99: (* normal operation *)
	(* only if input changes for an equivalent of min_ontime then change the output *)
	(* if there is a directional change then wait until last step is finished *)
	IF in < TIME_TO_REAL(min_ontime)/TIME_TO_REAL(max_runtime)/2 THEN val := 0;
	ELSIF in > 1 - TIME_TO_REAL(min_ontime)/TIME_TO_REAL(max_runtime)/2 THEN val := 1;
	ELSIF differ(LIMIT(0,in,1), val, TIME_TO_REAL(min_ontime) / TIME_TO_REAL(max_runtime)) OR in = 0 OR in = 1 THEN
		IF in < val AND NOT out1 THEN val := in;
		ELSIF in > val AND NOT out2 THEN val := in;
		END_IF;
	END_IF;

END_CASE;

(* output ramp generator *)
rout(in := val);
out1 := rout.busy AND rout.UD;
out2 := rout.busy AND NOT rout.UD;
pos := rout.out;

(* set the busy output and if busy goes low, then set the last time in order to check for min_offtime *)
IF NOT busy AND rout.busy THEN
	last := tn;
ELSIF busy AND NOT rout.busy THEN
	cal_timer := cal_timer + tx;
	last := tn;
END_IF;
busy := rout.busy;



(* revision history

19.10.2006	rev 1.1
	added security checks for end_switch to avoid overrun of the end_switch, hans

23.1.2007		rev 1.2
	deleted unused variables force_on and force_off

15.9.2007	hm	rev 1.3
	replaced Time() with T_PLC_MS for compatibility and performance reasons

*)

END_FUNCTION_BLOCK

// POUs/Mathematical/DIFFER
FUNCTION DIFFER : BOOL
VAR_INPUT
	in1 : REAL;
	in2 : REAL;
	X : REAL;
END_VAR


(*
version 1.1	16 mar 2008
programmer 	hugo
tested by		tobias

this function checks if in1 differs more then x from in2
the output is true if abs(in1-in2) > X

*)

DIFFER := ABS(in1 - in2) > X;

(* revision history
hm		8. oct 2006		rev 1.0
	original version

hm		16. mar 2008	rev 1.1
	improverd code for performance

*)

END_FUNCTION

// POUs/Time&Date/MULTIME
FUNCTION MULTIME : TIME
VAR_INPUT
	t : TIME;
	M : REAL;
END_VAR


(*
version 1.1	14 mar 2008
programmer 	hugo
tested by		tobias

multiplies a time by a real number and returns a time
*)

MULTIME := DWORD_TO_TIME(REAL_TO_DWORD(DWORD_TO_REAL(TIME_TO_DWORD(t))*M));

(* revision history
hm		2. oct 2006	rev 1.0
	original version

hm		14. mar 2008	rev 1.1
	rounded the result after the last digit

*)

END_FUNCTION

// POUs/Engineering/measurements/CALIBRATE
FUNCTION_BLOCK CALIBRATE
VAR_INPUT
	X : REAL;
	CO : BOOL;
	CS : BOOL;
END_VAR
VAR_INPUT CONSTANT
	Y_Offset : REAL;
	Y_Scale : REAL;
END_VAR
VAR_OUTPUT
	Y : REAL;
END_VAR
VAR RETAIN
	offset : REAL;
	Scale : REAL := 1.0;
END_VAR

(*
	version 1.3	11. mar. 2009
	programmer 	hugo
	tested BY		hans

Calibrate allows for offset and scale calibration of an analog input.
offset is calibrated to a stored reference Y_offset while CO is true.
after the offset is calibrated, scale can be calibrated to a reference value Y_scale while CS is true.
*)

(* check for calibration *)
IF CO THEN
	OFFSET := Y_Offset - X;
ELSIF CS THEN
	SCALE := Y_scale / (X + OFFSET);
END_IF;
(* calculate output *)
Y := (X + OFFSET) * SCALE;


(* revision history
hm 22.2.2007		rev 1.2
	changed VAR RETAIN PERSISTENT to VAR RETAIN for better compatibility
	wago lon contollers do not support persisitent

hm	11. mar. 2009	rev 1.3
	changed real constants to use dot syntax

*)

END_FUNCTION_BLOCK

// POUs/Engineering/signal processing/SCALE
FUNCTION SCALE : REAL
VAR_INPUT
	X : REAL;
	K : REAL;
	O : REAL;
	MX : REAL;
	MN : REAL;
END_VAR


(*
version 1.0	16. may. 2008
programmer 	hugo
tested by		tobias

Scale is used to translate an input x to output by the formula Y = X*K + O.
at the same time the output is limited to MN and MX.

*)

SCALE := LIMIT(MN, X * K + O, MX);


(* revision history
hm	16. may. 2008		rev 1.0
	original version
*)

END_FUNCTION

// POUs/Mathematical/functions/FT_RMP
FUNCTION_BLOCK FT_RMP
VAR_INPUT
	Rmp : BOOL := TRUE;
	in : REAL;
	KR : REAL;
	KF : REAL;
END_VAR
VAR_OUTPUT
	out : REAL;
	busy : BOOL;
	UD : BOOL;
END_VAR
VAR
	tx: TIME;
	last: TIME;
	init: BOOL;
END_VAR

(*
	version 1.4	25 jan 2008
	programmer 	oscat
	tested BY		oscat

this ramp function follows an input signal with a linear ramp up or down, the up or down speed can be set with KF and KR.
a K factor of 1 means 1 unit per second on the output. K factors can only be positive and not negative.
a busy output signals the ramp is running or busy false means the in value is present on the output.
a rmp input false means the output follows the input dierctly while a rmp = true means the output follows the input with a ramp.
a updn output signal the directon of the ramp (up or down).

*)

(* read system time *)
tx := DWORD_TO_TIME(T_PLC_MS()) - last;

IF NOT init THEN
	init := TRUE;
	last := tx;
	tx := t#0s;
	out := in;
END_IF;
IF NOT rmp THEN
	out := in;
	busy := FALSE;
ELSIF out > in THEN
	(* ramp down *)
	out := out - TIME_TO_REAL(tx) * 0.001 * KF;
	out := MAX(in, out);
ELSIF out < in THEN
	(* ramp up *)
	out := out + TIME_TO_REAL(tx) * 0.001 * KR;
	out := MIN(in, out);
END_IF;

(* set busy and dir flags *)
IF out < in THEN
	busy := TRUE;
	ud := TRUE;
ELSIF out > in THEN
	busy := TRUE;
	ud := FALSE;
ELSE
	busy := FALSE;
END_IF;
last := last + tx;


(* revision history:

hm 8.10.2006			rev 1.1
	added ud output

hm 12. feb 2007		rev 1.2
	added init variable and corrected a possible startup problem

hm	17. sep 2007	rev 1.3
	replaced time() with t_plc_ms() for compatibility reasons

hm	25. jan 2008	rev 1.4
	performance improvements
	allow KR and KF to be 0
*)

END_FUNCTION_BLOCK

// POUs/Building/actuators/ACTUATOR_A
FUNCTION_BLOCK ACTUATOR_A
VAR_INPUT
	I1 : BYTE;
	IS : BOOL;
	I2 : BYTE;
	RV : BOOL;
	DX : BOOL;
END_VAR
VAR_INPUT CONSTANT
	RUNTIME : TIME;
	SELF_ACT_TIME : TIME;
	OUT_MIN : WORD;
	OUT_MAX : WORD;
END_VAR
VAR_OUTPUT
	Y : WORD;
END_VAR
VAR
	timer : CYCLE_4;
	dx_edge: BOOL;
END_VAR


(*
version 1.0 8. nov. 2008	
programmer 	hugo
tested by	oscat

ACTUATOR_A drives any valve or similar with 0 - 255 continuous control input.
 
*)

(* run the system timer, if self_act_time = t#0s then state is set to 0 *)
timer(T0 := RUNTIME, T1 := RUNTIME, T3 := SELF_ACT_TIME, sl := DX AND NOT dx_edge, sx := 0, S0 := SELF_ACT_TIME > t#0s);
dx_edge := dx;

CASE timer.STATE OF
	0: 	(* self act min value *)
		Y := OUT_MIN;
	1:	(* self_act max value *)
		Y := OUT_MAX;
	3:	(* normal operation *)
		IF rv THEN
			Y := OUT_MAX - (OUT_MAX - OUT_MIN) * SEL(IS, I1, I2) / 255;
		ELSE
			Y := (OUT_MAX - OUT_MIN) * SEL(IS, I1, I2) / 255 + OUT_MIN;
		END_IF;
END_CASE;




(*
hm 	8. nov. 2008	rev 1.0
	original version

*)

END_FUNCTION_BLOCK

// POUs/Logic/generators/CYCLE_4
FUNCTION_BLOCK CYCLE_4
VAR_INPUT
	E : BOOL := TRUE;
	T0, T1, T2, T3 : TIME;
	S0 : BOOL;
	SX : INT;
	SL : BOOL;
END_VAR
VAR_OUTPUT
	STATE : INT;
END_VAR
VAR
	tx : TIME;
	last : TIME;
	init: BOOL;
END_VAR


(*
version 1.0	
programmer 	hugo
tested by	oscat


 
*)

(* read system timer *)
tx := DWORD_TO_TIME(T_PLC_MS());
(* init on first cycle *)
IF NOT init THEN
	init := TRUE;
	last := tx;
END_IF;

IF E THEN
	IF SL THEN
		(* when sx > 0 then the state sx is forced to start *)
		state:= LIMIT(0,SX,3);
		last := tx;
		(* this is to avoid to reset sx from the calling programm it does work fine on codesys but i am not sure about other systems, because we are writing to an input *)
		SL := FALSE;
	ELSE
		CASE state OF
			0 :	(* wait for T0 and switch to next cycle *)
				IF tx - last >= T0 THEN
					state := 1;
					last := tx;
				END_IF;
			1 : (* wait for T1 over 1st cycle *)
				IF tx - last >= T1 THEN
					state := 2;
					last := tx;
				END_IF;
			2 : (* wait for T1 over 1st cycle *)
				IF tx - last >= T2 THEN
					state := 3;
					last := tx;
				END_IF;
			3 : (* wait for T2 over 2nd cycle *)
				IF tx - last >= T3 THEN
					IF S0 THEN State := 0; END_IF; (* if S0 is false, the sequence stops at state 3 *)
					last := tx;
				END_IF;
		END_CASE;
	END_IF;
ELSE
	state := 0;
	last := tx;
END_IF;



(*
hm	3. nov. 2008	rev 1.0
	original version

*)

END_FUNCTION_BLOCK

// POUs/Building/actuators/ACTUATOR_COIL
FUNCTION_BLOCK ACTUATOR_COIL
VAR_INPUT
	IN : BOOL;
END_VAR
VAR_INPUT CONSTANT
	self_act_cycle : TIME := t#10d;
	self_act_time : TIME := t#1s;
END_VAR
VAR_OUTPUT
	OUT :BOOL;
	STATUS : BYTE;
END_VAR
VAR
	last : DWORD;
	init: BOOL;
	tx: DWORD;
	now: DWORD;
END_VAR


(*
version 1.0	1. jun. 2008
programmer 	hugo
tested by		tobias

this is an intelligent actuator interface for any coil actuator.
the coil actuator can only switch on/off.
coil actuators like vents can get stuck if they are not u8sed for a long time and need to be autoactivated on ce in a while.

*)

(* read system time *)
now := T_PLC_MS();

(* initialize for first cycle *)
IF NOT init THEN
	last := now;
	init := TRUE;
ELSIF IN THEN
	OUT := TRUE;
	STATUS := 101; (* activated by input *)
	LAST := now;
ELSE
	OUT := FALSE;
	STATUS := 100; (* disabled *)
	(* now we need to check for self activation *)
	tx := now - last;
	IF (self_act_cycle > T#0s) AND (tx >= TIME_TO_DWORD(self_act_cycle)) THEN
		OUT := TRUE;
		STATUS := 102; (* auto activation *)
		IF tx >= TIME_TO_DWORD(self_act_cycle + self_act_time) THEN
			last := now;
			OUT := FALSE;
			STATUS := 100; (* idle *)
		END_IF;
	END_IF;
END_IF;



(*
revision history:

hm		1. jun. 2008 	rev 1.0
	original version

*)

END_FUNCTION_BLOCK

// POUs/Building/actuators/ACTUATOR_PUMP
FUNCTION_BLOCK ACTUATOR_PUMP
VAR_INPUT
	IN : BOOL;
	MANUAL : BOOL;
	RST : BOOL;
END_VAR
VAR_INPUT CONSTANT
	MIN_ONTIME : TIME := t#10s;
	MIN_OFFTIME : TIME := t#10s;
	RUN_EVERY : TIME := t#10000m;
END_VAR
VAR_OUTPUT
	PUMP : BOOL;
END_VAR
VAR_IN_OUT
	RUNTIME : UDINT;
	CYCLES : UDINT;
END_VAR
VAR
	tx : TIME;
	last_change : TIME;
	meter : ontime;
	old_man : BOOL;
	init: BOOL;
END_VAR

(*
version 1.4		21. oct. 2008
programmer 		oscat
tested BY		oscat

actuator_pump is a pump interface which can be controlled by an input in and an input manual.
in or manual high turns the pump output on.
a rst input is used to reset the runtime counters.
when the pump was not active for a time run_every the actuator turns on the pump automatically for min_ontime.
two setup variables min_ontime and min_offtime guarantee a minimum runtime and offtime of the pump.
the units are hours and the output type is real to prevent from overfow.

*)

tx := DWORD_TO_TIME(T_PLC_MS());

IF NOT init THEN
	init := TRUE;
	last_change := tx;
ELSIF rst THEN
	rst := FALSE;
	runtime := 0;
	cycles := 0;
ELSIF manual AND NOT pump AND NOT old_man THEN
	last_change := tx;
	pump := TRUE;
ELSIF NOT manual AND old_man AND pump AND NOT in THEN
	last_change := tx;
	pump := FALSE;
ELSIF in AND NOT pump AND tx - last_change >= min_offtime THEN
	last_change := tx;
	pump := TRUE;
ELSIF pump AND NOT in AND NOT manual AND tx - last_change >= min_ontime THEN
	last_change := tx;
	pump := FALSE;
ELSIF NOT pump AND (tx - last_change >= run_every) AND (run_every > T#0s) THEN
	last_change := tx;
	pump := TRUE;
END_IF;

meter(in := pump, seconds := runtime, cycles := cycles);
old_man := manual;



(*
hm	27.12.2006		rev 1.1
	fixed a failure while the pump would run for tmin after startup.

hm	15.9.2007		rev 1.2
	replaced Time() with T_PLC_MS for compatibility and performance reasons

hm	13. oct. 2008	rev 1.3
	auto activation can now be disabled when run_every = t#0s

hm	21. oct. 2008	rev 1.4
	changed to use ontime rev 2.0

*)

END_FUNCTION_BLOCK

// POUs/Engineering/automation/MANUAL
FUNCTION MANUAL : BOOL
VAR_INPUT
	IN : BOOL;
	ON : BOOL;
	OFF : BOOL;
END_VAR


(*
version 1.0	21. nov. 2008
programmer 	hugo
tested by	oscat

MANUAL is a manual override for digital signals.
when on and off = FALSE, the output follows IN.
ON = TRUE forces the output high, and OFF = TRUE forces the output low.


*)

MANUAL := NOT OFF AND (IN OR ON);



(* revision history
hm	21. nov 2008	rev 1.0
	original version


*)

END_FUNCTION

// POUs/Engineering/signal processing/OVERRIDE
FUNCTION OVERRIDE : REAL
VAR_INPUT
	X1, X2, X3 : REAL;
	E1 : BOOL;
	E2 : BOOL;
	E3 : BOOL;
END_VAR


(*
version 1.0	4 nov 2007
programmer 	oscat
tested by	tobias

OVERRIDE deliveres the maximum absolute value of the 3 inputs X1, X2 and X3.
with the inputs E1, E2 and E3 each of the 3 inputs can be turned on or off.

*)

IF E1 THEN OVERRIDE := X1; END_IF;
IF E2 AND ABS(x2) > ABS(OVERRIDE) THEN OVERRIDE := X2; END_IF;
IF E3 AND ABS(x3) > ABS(OVERRIDE) THEN OVERRIDE := X3; END_IF;

(* revision history
hm	4.11.2007		rev 1.0
	original version

*)

END_FUNCTION

// POUs/Logic/generators/TMIN
FUNCTION_BLOCK TMIN
VAR_INPUT
	IN : BOOL;
	PT : TIME;
END_VAR
VAR_OUTPUT
	Q : BOOL;
END_VAR
VAR
	pm : TP;
END_VAR

(*
version 1.0	21. jul. 2008
programmer 	hugo
tested by	oscat

Q of tMIN will follow IN except that it forces a minimum ontime for the output Q.

*)

pm(in := IN, PT := PT);
Q := IN OR pm.Q;


(* revision history
hm	21. jul. 2008	rev 1.0
	original version

*)

END_FUNCTION_BLOCK

// POUs/Building/actuators/ACTUATOR_UD
FUNCTION_BLOCK ACTUATOR_UD
VAR_INPUT
	UD : BOOL;
	ON : BOOL;
	Manual : BOOL;
	Up : BOOL;
	Dn : BOOL;
	off : BOOL;
	YUP_in : BOOL;
	YDN_in : BOOL;
END_VAR
VAR_INPUT CONSTANT
	TON : TIME;
	TOFF : TIME;
	out_return : BOOL;
END_VAR
VAR_OUTPUT
	Yup : BOOL;
	Ydn : BOOL;
	status : BYTE;
END_VAR
VAR
	tx : TIME;
	last : TIME;
	init: BOOL;
END_VAR

(*
version 1.3	17. oct. 2008
programmer 	hugo
tested by		tobias

out_ud is a up/dn or Right/left locked output driver.
it can be controlled by automatic inputs UD and ON as well as manual inputs for up and dn.
a security input to shut off at any time is prvided by the off input.
two time set inputs ton and toff specify a minimum on time for outputs and a minimum off time before the next output can become active.
the module assures that only one output can be active at any time.
for higher security pls make sure you use hardware locking of the outputs to prevent from defective wiring or outputs.
further security is provided b feedback inputs Yup_in and Ydn_in which are separate inputs for the output signal, if these inputs are not available 
pls connect them directly to Yup and Ydn.
manual mode will override automatic mode by setting the manual input high.
a status output will be 0 for normal operation or 1 - 99 for error reporting and 101 - 199 for status reporting
The status output is ESR comptible.
*)

(* read system time *)
tx := DWORD_TO_TIME(T_PLC_MS());

IF NOT init THEN
	(* INITIALIZATION AT FIRST CALL *)
	last := tx;
	init := TRUE;
ELSIF off THEN
	(* emergency shut off detected *)
	Yup := FALSE;
	ydn := FALSE;
	last := tx;
	status := 101;

(* Watch FOR MIN TON TIME *)
ELSIF ((Yup OR Ydn) AND tx - last < Ton) THEN
	RETURN;
ELSIF NOT yup AND NOT ydn AND tx - last < toff THEN
	RETURN;

(* manual operation *)
ELSIF manual THEN
	status := 102;
	(* directional chage set both outs 0 first *)
	IF yup AND NOT up OR ydn AND NOT dn THEN
		ydn := FALSE;
		yup := FALSE;
		last := tx;
	(* manual up operation *)
	ELSIF UP AND NOT DN AND NOT OFF THEN
		Ydn := FALSE;
		Yup := TRUE;
		last := tx;
		status := 103;
	(* manual down operation *)
	ELSIF DN AND NOT UP AND NOT OFF THEN
		Yup := FALSE;
		Ydn := TRUE;
		last := tx;
		status := 104;
	(* maual mode but no up or down *)
	ELSE
		IF YUP OR YDN THEN LAST := tx; END_IF;
		Yup := FALSE;
		ydn := FALSE;
	END_IF;

(* automatic operation *)
ELSE
	(* directional change set outputs low first *)
	IF yup AND NOT ud OR ydn AND UD THEN
		yup := FALSE;
		ydn := FALSE;
		last := tx;
	(* automatic up operation *)
	ELSIF Ud AND on AND NOT OFF THEN
		Ydn := FALSE;
		Yup := TRUE;
		last := tx;
		status := 111;

	(* automatic down operation *)
	ELSIF NOT UD AND on AND NOT OFF THEN
		Yup := FALSE;
		Ydn := TRUE;
		last := tx;
		status := 112;
	(* standby mode *)
	ELSE
		IF Yup OR Ydn THEN last := tx; END_IF;
		Yup := FALSE;
		Ydn := FALSE;
		status := 110;
	END_IF;
END_IF;

(* make sure Yup and Ydn are never on at the same time *)
IF Ydn AND Yup_in AND out_return THEN
	Ydn := FALSE;
	status := 1;
END_IF;
IF Yup AND Ydn_in AND out_return THEN
	Yup := FALSE;
	status := 2;
END_IF;



(* revision history
hm 22. jan 2007	rev 1.1
	added status output
	changed inputs ton, toff to config variables
	added config var out_return to enable yup_in and Ydn_in
	manual mod will override automatic mode 

hm	15.9.2007	rev 1.2
	replaced Time() with T_PLC_MS for compatibility and performance reasons

hm	17. oct. 2008	rev 1.3
	deleted unnecessary initialization with 0
*)

END_FUNCTION_BLOCK

// POUs/Mathematical/AGDF
FUNCTION AGDF : REAL
VAR_INPUT
	X : REAL;
END_VAR


(*
version 1.1	10. mar. 2009
programmer 	hugo
tested by		tobias

this function calculates the inverse Gudermannian function.

*)

AGDF := LN((1.0 + SIN(X)) / COS(X));

(* comment
the current implementation gives sufficient accuracy only up to X = 1.57 or an output > 10.
is X closer to PI/2 then the function is more and more unreliable
*)



(* revision history
hm	27. apr. 2008	rev 1.0
	original version

hm	10. mar. 2009	rev 1.1
	real constants updated to new systax using dot

*)

END_FUNCTION

// POUs/Engineering/signal processing/AIN
FUNCTION AIN : REAL
VAR_INPUT
	in : DWORD;
END_VAR
VAR_INPUT CONSTANT
	Bits : BYTE;
	sign : BYTE := 255;
	low : REAL;
	high : REAL := 10.0;
END_VAR
VAR CONSTANT
	ff : DWORD := 16#FFFFFFFF;
END_VAR
VAR
	temp1 : DWORD;
	temp2 : DWORD;
	sx : BOOL;
END_VAR

(*
version 1.5	16 mar 2008
programmer 	oscat
tested by		tobias

Ain converts signals from A/D converters or other digital sources to an internal real value
the lowest number of bits are extracted from the input word and the sign will be extracted if available separately.
the output signal is then conditioned to range from low to high values for a 0 to max value on the analog inputs:
for example a 15bit input (bits := 12) with sign at bit 15 (0..15) will deliver 0.0 (low value at 0) for an input value of 2#0000_0000_0000
an input value of 2#1111_1111_1111 will deliver 10.0 on the output (high value set to 10).

*)

(* extract the sign bit *)
IF sign < 32 THEN
	temp1 := SHR(in,sign);
	sx := temp1.0;
ELSE
	sx := FALSE;
END_IF;
temp1 := SHR(ff, 32-bits);
temp2 := in AND temp1;
AIN := (high - low) * DWORD_TO_REAL(temp2) / DWORD_TO_REAL(temp1) + low;
IF sx THEN AIN := -AIN; END_IF;

(* revision history
hm 18.8.2006	rev 1.1
	fixed an error with low value negative and high value 0.

hm 19.1.2007	rev 1.2
	fixed an error with sign bit.

hm	13.9.2007	rev 1.3
	changed code to avoid warning under codesys 2.8.1

hm	2. dec 2007	rev 1.4
	changed code for better performance

hm	16. mar 2008	rev 1.5
	added type conversions to avoid warnings under codesys 30
*)

END_FUNCTION

// POUs/Engineering/signal processing/AIN1
FUNCTION_BLOCK AIN1
VAR_INPUT
	in : DWORD;
END_VAR
VAR_INPUT CONSTANT
	sign_bit : INT := 255;
	error_bit : INT := 255;
	error_code_en : BOOL;
	error_code : DWORD;
	overflow_bit : INT := 255;
	overflow_code_en : BOOL;
	overflow_code : DWORD;
	Bit_0 : INT;
	Bit_N : INT := 31;
	out_min : REAL;
	out_max : REAL := 10.0;
	code_min : DWORD;
	code_max : DWORD := 16#FFFFFFFF;
	error_output : REAL;
	overflow_output : REAL := 10.0;
END_VAR
VAR_OUTPUT
	out : REAL;
	sign : BOOL;
	error : BOOL;
	overflow : BOOL;
END_VAR
VAR
	tB: DWORD;
END_VAR

(*
version 1.3	10. mar. 2009
programmer 	oscat
tested by		tobias

Ain1 converts signals from A/D converters or other digital sources to an internal real value.

*)

(* extract error bit *)
error := ((SHR(in,error_bit) AND 16#0000_0001) = 1) OR (error_code_en AND error_code = in);
IF error THEN
	out := error_output;
	RETURN;
END_IF;

(* strip off the data input *)
tb := SHR(SHL(in, 31 - bit_N), 31 - bit_N + Bit_0);

(* extract overflow bit *)
overflow := ((SHR(in,overflow_bit) AND 16#0000_0001) = 1) OR (overflow_code_en AND overflow_code = in) OR (tb < code_min OR tb > code_max);
IF overflow THEN
	out := overflow_output;
	RETURN;
END_IF;

(* extract sign bit *)
sign := (SHR(in,sign_bit) AND 16#0000_0001) = 1;

(* convert in to out *)
out := (DWORD_TO_REAL(tb - code_min) * (out_max - out_min) / DWORD_TO_REAL(code_max - code_min) + out_min);
IF sign THEN out := out * -1.0; END_IF;



(* revision history
hm	23. feb 2008	rev 1.0
	original version

hm	16. mar 2008	rev 1.1
	added type conversions to avoid warnngs under codesys 30

hm	22. apr. 2008	rev 1.2
	corrected error in formula when code_min was set
	corrected error when sign bit was used
	optimized code for better performance

hm	10. mar. 2009	rev 1.3
	real constants updated to new systax using dot

*)

END_FUNCTION_BLOCK

// POUs/Building/HLK/AIR_DENSITY
FUNCTION AIR_DENSITY : REAL
VAR_INPUT
	T : REAL;
	P : REAL;
	RH : REAL;
END_VAR
VAR CONSTANT
	RL : REAL := 287.05;
	RX : REAL := 3.773319E-3;
END_VAR


(*
version 1.3	13. mar. 2009
programmer 	hugo
tested by		tobias

this function calculates the air density between 0 and 100 deg C

*)

AIR_DENSITY := phys.PN * (1.0 - RH * SDD(T, TRUE) * RX / P) / (RL * ( T - phys.T0));

(* original code used for rev 1.0

SDD := SDD(T,FALSE);
RF := RL / (1- RH*SDD/P*RX);
Air_density := P / (RF * (T-TK));

*)

(* revision history

hm	29.10.2007	rev 1.0
	original version

hm	4.12.2007		rev 1.1
	changed code for better performance

hm	18. oct. 2008	rev 1.2
	using phys constants

hm	13. mar. 2009	rev 1.3
	real constants updated to new systax using dot

*)

END_FUNCTION

// POUs/Building/HLK/SDD
FUNCTION SDD : REAL
VAR_INPUT
	T : REAL;
	ICE: BOOL;
END_VAR


(*
version 1.1	2 dec 2007
programmer 	hugo
tested by		tobias

this function calculates the vapor saturation pressure for moist Air over ice or water

*)

IF ice THEN
	SDD := 611.153 * EXP(22.4433 * T / (272.186 + T));
ELSE
	SDD := 611.213 * EXP(17.5043 * T / (241.2 + T));
END_IF;



(* revision history

hm 29 oct 2007		rev 1.0
	original version

hm	2. dec 2007		rev 1.1
	changed code for better performance
*)

END_FUNCTION

// POUs/Engineering/conversion/PRESSURE
FUNCTION_BLOCK PRESSURE
VAR_INPUT
	mws : REAL;
	torr : REAL;
	att : REAL;
	atm : REAL;
	pa : REAL;
	bar : REAL;
END_VAR
VAR_OUTPUT
	Ymws : REAL;
	Ytorr : REAL;
	Yatt : REAL;
	Yatm : REAL;
	Ypa : REAL;
	Ybar : REAL;
END_VAR


(*
version 1.1	11. mar. 2009
programmer 	hugo
tested by		oscat

this function converts different pressure units
any unused input can simply be left open.
different inputs connected at the same time will be added up.
*)

Ybar := bar +
		pa * 1.0E-5 +
		0.980665 * att +
		1.01325 * atm +
		0.001333224 * torr +
		0.0980665 * mws;
Ymws := ybar * 10.1971621297793;
Ytorr := ybar * 750.0615050434140;
Yatt := ybar * 1.0197162129779;
yatm := ybar * 0.9869232667160;
Ypa := ybar * 100000.0;


(*
Druck, Pascal Pa 1 Pa = 1 N/m2 = 1 kg/(s2 E m) . 0,75 E 10.2 mmHg
mechanische 1 MPa = 1 N/mm2 . fur Festigkeitsangaben
Spannung Bar bar 1 bar = 105 Pa = 103 mbar = 105 kg/(s2 E m)
Millimeter- mmHg 1 mmHg = 133,322 Pa = 1,333 22 mbar
Quecksilbersaule . nur in Heilkunde zulassig
physik. Atmosphare atm 1 atm = 1,013 25 bar
techn. Atmosphare at 1 at = 1 kp/cm2 = 0,980665 bar
Torr Torr 1 Torr = (101325/760) Pa = 1,333224 mbar
Meter-Wassersaule mWS 1 mWS = 9806,65 Pa = 98,0665 mbar
psi lbf/in2 1 lbf/in2 = 68,947 57 mbar = 6894,757 Pa

*)

(* revision history

hm	27. mar. 2007	rev 1.0
	original version

hm	11. mar. 2009	rev 1.1
	improved code

*)

END_FUNCTION_BLOCK

// POUs/Mathematical/DEG
FUNCTION DEG : REAL
VAR_INPUT
	rad : REAL;
END_VAR


(*
version 1.2	10. mar. 2009
programmer 	hugo
tested by		tobias

this function converts degrees into Radiant
execution time on wago 750 - 841 =  10  us
*)

DEG := MODR(57.29577951308232 * RAD, 360.0);

(* revision history
hm	4. aug 2006	rev 1.0
	original version

hm 16. oct 2007	rev 1.1
	added modr statement which prohibits deg to become bigger than 360

hm	10. mar. 2009	rev 1.2
	real constants updated to new systax using dot
*)

END_FUNCTION

// POUs/Mathematical/RAD
FUNCTION RAD : REAL
VAR_INPUT
	deg : REAL;
END_VAR


(*
version 1.2	18. oct. 2008
programmer 	hugo
tested by	tobias

this function converts Radiant to degrees

*)

RAD := MODR(0.0174532925199433 * DEG, math.PI2);

(* revision history
hm	4. aug 2006		rev 1.0
	original version

hm 	16. oct 2007	rev 1.1
	added modr statement which prohibits rad to become bigger than 2PI

hm	18. oct 2008	rev 1.2
	using math constants

*)

END_FUNCTION

// POUs/Building/HLK/AIR_ENTHALPY
FUNCTION AIR_ENTHALPY : REAL
VAR_INPUT
	T : REAL;
	RH : REAL;
END_VAR
VAR CONSTANT
	CPL : REAL := 1.00482;
	CW : REAL := 1.86;
	LH : REAL := 2500.78;
END_VAR


(*
version 1.1	2 nov 2007
programmer 	hugo
tested by		tobias

this function calculates the enthalpy for humid air between 0 and 100 deg C

*)

AIR_ENTHALPY := CPL * T + (CW * T + LH) * DEW_CON(RH,T);

(* revision history

hm	31.10.2007	rev 1.0
	original version

hm	2.11.2007		rev 1.1
	deleted unused variable RF

hm	2.12.2007		rev 1.2
	changed code for better performance
*)

END_FUNCTION

// POUs/Building/HLK/DEW_CON
FUNCTION DEW_CON : REAL
VAR_INPUT
	RH : REAL;
	T : REAL;
END_VAR


(*
version 1.5	13. mar. 2009
programmer 	hugo
tested by		oscat

this function calculates the water concentratin in air for a given temperature and relative humidity.
the output states the concentration of water vapor in air in Gramms / qubic meter.

*)

(*	this code is good to read but need to be improoved
	SDD := 6.1078*EXPT(10,(a*T)/(b+T));
	DD := RH/100 * SDD;
	V := LOG(DD/6.1078);
	TD := b*V/(a-v);
	dew_con := 0.1 * mw / RU * DD / (T - TK);
*)
IF RH > 0.0 THEN
	DEW_CON := 2.166824303E-2 * RH * SDD(T,FALSE)  / (T - phys.T0);
END_IF;

(*
Bezeichnungen:
r = relative Luftfeuchte
T = Temperatur in °C
TK = Temperatur in Kelvin (TK = T + 273.15)
TD = Taupunkttemperatur in °C
DD = Dampfdruck in hPa
SDD = Sättigungsdampfdruck in hPa

Parameter:
a = 7.5, b = 237.3 für T >= 0
a = 7.6, b = 240.7 für T < 0 über Wasser (Taupunkt)
a = 9.5, b = 265.5 für T < 0 über Eis (Frostpunkt)

R* = 8314.3 J/(kmol*K) (universelle Gaskonstante)
mw = 18.016 kg (Molekulargewicht des Wasserdampfes)
AF = absolute Feuchte in g Wasserdampf pro m3 Luft

Formeln:

   1. SDD(T) = 6.1078 * 10^((a*T)/(b+T))
   2. DD(r,T) = r/100 * SDD(T)
   3. r(T,TD) = 100 * SDD(TD) / SDD(T)
   4. TD(r,T) = b*v/(a-v) mit v(r,T) = log10(DD(r,T)/6.1078)
   5. AF(r,TK) = 10^5 * mw/R* * DD(r,T)/TK; AF(TD,TK) = 10^5 * mw/R* * SDD(TD)/TK 

*)

(* revision history

hm 29 apr 2007	rev 1.0
	original version

hm	13.sep 2007	rev 1.1
	improoved coding for speed
	deleted unused variabled SDD,DD,V, TD

hm	2. dec 2007	rev 1.2
	changed code for better performance
	output is now in Gramms / Qubic meter

hm	14. oct. 2008	rev 1.3
	performance improvement

hm	18. oct. 2008	rev 1.4
	using phys constants

hm	13. mar. 2009	rev 1.5
	improved code
*)

END_FUNCTION

// POUs/Engineering/conversion/TEMPERATURE
FUNCTION_BLOCK TEMPERATURE
VAR_INPUT
	K : REAL;
	C : REAL := -273.15;
	F : REAL := -459.67;
	Re : REAL := -218.52;
	Ra : REAL;
END_VAR
VAR_OUTPUT
	YK : REAL;
	YC : REAL;
	YF : REAL;
	YRe : REAL;
	YRa : REAL;
END_VAR


(*
version 1.0	21 feb 2008
programmer 	hugo
tested by	oscat

this function converts different temperature units
any unused input can simply be left open.
different inputs connected at the same time will be added up.

*)

YK := K + (C + 273.15) + (F + 459.67) * 0.555555555555 + (Re * 1.25 + 273.15) + (Ra * 0.555555555555);
YC := YK -273.15;
YF := YK * 1.8 - 459.67;
YRe := (YK - 273.15) * 0.8;
YRa := YK * 1.8;


(* revision history
hm	21. feb. 2008	rev 1.0
	original version

*)

END_FUNCTION_BLOCK

// POUs/Engineering/measurements/ALARM_2
FUNCTION_BLOCK ALARM_2
VAR_INPUT
	X : REAL;
	LO_1 : REAL;
	HI_1 : REAL;
	LO_2 : REAL;
	HI_2 : REAL;
	HYS : REAL;
END_VAR
VAR_OUTPUT
	Q1_LO : BOOL;
	Q1_HI : BOOL;
	Q2_LO : BOOL;
	Q2_HI : BOOL;
END_VAR
VAR
	tmp: REAL;
END_VAR

(*
	version 1.1	11. mar. 2009
	programmer 	hugo
	tested BY		tobias

ALARM_2 will check two pairs of limits and signal when the input is above or below a set limit.
with the input HYS a hysteresis can be defined for all limits. 

*)

tmp := X - Hys * 0.5;
IF tmp > LO_1 THEN Q1_LO := FALSE; END_IF;
IF tmp > LO_2 THEN Q2_LO := FALSE; END_IF;
IF tmp > HI_1 THEN Q1_HI := TRUE; END_IF;
IF tmp > HI_2 THEN Q2_HI := TRUE; END_IF;
tmp := tmp + hys;
IF tmp < LO_1 THEN Q1_LO := TRUE; END_IF;
IF tmp < LO_2 THEN Q2_LO := TRUE; END_IF;
IF tmp < HI_1 THEN Q1_HI := FALSE; END_IF;
IF tmp < HI_2 THEN Q2_HI := FALSE; END_IF;



(* revision history
hm	19. may. 2008		rev 1.0
	original version

hm	11. mar. 2009	rev 1.1
	improved code
*)

END_FUNCTION_BLOCK

// POUs/Engineering/signal processing/AOUT
FUNCTION AOUT : DWORD
VAR_INPUT
	in : REAL;
END_VAR
VAR_INPUT CONSTANT
	Bits : BYTE;
	sign : BYTE := 255;
	low : REAL;
	high : REAL := 10.0;
END_VAR
VAR CONSTANT
	ff : DWORD := 2#1;
END_VAR
VAR
	in2 : REAL;
	sx : BOOL;
END_VAR

(*
version 1.4	23 feb 2008
programmer 	oscat
tested by		tobias

this module conditions an internal real value for D/A converter.
Aout converts and internal real value to a word for an D/A converter or other output devices.
The input value is converted to a n-bit wide output and a sign bit is set separately as specified.
the outout min value is set for the specified min input value and the max output is set for the max input value.
an input higher or lower then the max or min value will set the respective max or min value or the output.


*)

(* if sign bit is defined *)
IF sign < 32 THEN
	sx := sign_R(in);
	in2 := ABS(in);
ELSE
	in2 := in;
END_IF;

(* begrenze in auf die zulässigen werte *)
in2 := LIMIT(low, in2, high);

(* Berechne den Ausgangswert *)
Aout := REAL_TO_DWORD((in2 - low) / (high - low) * DWORD_TO_REAL(SHL(ff,bits) -1));
IF sx THEN Aout := SHL(ff,sign) OR Aout; END_IF;

(*
revision history

hm 18.1.2007		rev 1.1
	renamed Modul to aout.
	changed Output to 32 Bit max.
	corrected error with sign bit.

hm	13.9.2007		rev 1.2
	changed code to avoid warning under codesys 2.8.1

hm	2. dec 2007		rev 1.3
	changed code for better performance

hm	23. feb 2008	rev 1.4
	changed code for better performance
*)

END_FUNCTION

// POUs/Mathematical/SIGN_R
FUNCTION SIGN_R : BOOL
VAR_INPUT
	in : REAL;
END_VAR


(*
version 1.4	10. mar. 2009
programmer 	hugo
tested by		tobias

this function return true if the real input is negative

*)

SIGN_R := in < 0.0;


(* revision history
hm 19.1.2007	rev 1.1
	changed method of function for better compatibility to other systems

hm	1.12.2007	rev 1.2
	changed code to improve performance

hm	14. jun. 2008	rev 1.3
	improved performace

hm 10. mar. 2009	rev 1.4
	real constants updated to new systax using dot																																																																																																																																																																																																																																																																																																																																																																																																																																																																																																																																																																																																																																																																																																																																																																																																																																																																																																																																																																																																																																																											

*)

END_FUNCTION

// POUs/Engineering/signal processing/AOUT1
FUNCTION AOUT1 : DWORD
VAR_INPUT
	in : REAL;
END_VAR
VAR_INPUT CONSTANT
	Bit_0 : INT;
	Bit_N : INT := 31;
	sign : INT := 255;
	low : REAL;
	high : REAL := 10.0;
END_VAR
VAR CONSTANT
	ff : DWORD := 2#1;
END_VAR
VAR
	sx: BOOL;
	in2 : REAL;
END_VAR

(*
version 1.0	23 feb 2008
programmer 	oscat
tested by		tobias

this module conditions an internal real value for a D/A converter.

*)

(* if sign bit is defined *)
IF sign < 32 THEN
	sx := SIGN_R(in);
	in2 := ABS(in);
ELSE
	in2 := in;
END_IF;

(* begrenze in auf die zulässigen werte *)
in2 := LIMIT(low, in2, high);

(* Berechne den Ausgangswert *)
AOUT1 := SHL(REAL_TO_DWORD((in2 - low) / (high - low) * DWORD_TO_REAL(SHL(ff,bit_n - Bit_0 + 1) -1)),Bit_0);
IF sx THEN AOUT1 := SHL(ff,sign) OR AOUT1; END_IF;


(* revision history
hm	23. feb 2008	rev 1.0
	original version

*)

END_FUNCTION

// POUs/Mathematical/Array/ARRAY_GAV
FUNCTION ARRAY_GAV : REAL
VAR_INPUT
	pt : POINTER TO ARRAY[0..32000] OF REAL;
	size : UINT;
END_VAR
VAR
	i: UINT;
	stop: UINT;
END_VAR

(*
version 1.1	10. mar. 2009
programmer 	hugo
tested by		tobias

this function will calculate the geometric average of a given array.
the function needs to be called:	array_avg(adr("array"),sizeof("array"));
because this function works with pointers its very time efficient and it needs no extra memory.

*)

stop := SHR(size,2)-1;
ARRAY_GAV := 1.0;
FOR i := 0 TO stop DO
	IF pt^[i] > 0.0 THEN
		ARRAY_GAV := ARRAY_GAV * pt^[i];
	ELSE
		ARRAY_GAV := 0.0;
		RETURN;
	END_IF;
END_FOR;
ARRAY_GAV := SQRTN(ARRAY_GAV,UINT_TO_INT(stop)+1);


(* revision history
hm	2. apr 2008	rev 1.0
	original version

hm	10. mar. 2009	rev 1.1
	real constants updated to new systax using dot

*)

END_FUNCTION

// POUs/Mathematical/SQRTN
FUNCTION SQRTN : REAL
VAR_INPUT
	X : REAL;
	N : INT;
END_VAR


(*
version 1.3	10. mar. 2009
programmer 	hugo
tested by		tobias

this function calculates the nth root function of X according to the formula sqrtn = x^(1/n).

*)

IF N > 0 THEN
	SQRTN := EXP(LN(x) / INT_TO_REAL(n));
ELSE
	SQRTN := 0.0;
END_IF;


(* revision history
hm		12 jan 2007	rev 1.0
	original version

hm		2. dec 2007	rev 1.1
	changed code for better performance

hm		11. mar 2008	rev 1.2
	added result 0 for compatibility reasons

hm 10. mar. 2009	rev 1.3
	added type conversions for compatibility reasons																																																																																																																																																																																																																																																																																																																																																																																																																																																																																																																																																																																																																																																																																																																																																																																																																																																																																																																																																																																																																																																									

*)

END_FUNCTION

// POUs/Mathematical/Array/ARRAY_HAV
FUNCTION ARRAY_HAV : REAL
VAR_INPUT
	pt : POINTER TO ARRAY[0..32000] OF REAL;
	size : UINT;
END_VAR
VAR
	i: UINT;
	stop: UINT;
END_VAR

(*
version 1.1	10. mar. 2009
programmer 	hugo
tested by		tobias

this function will calculate the harmonic average of a given array.
the function needs to be called:	array_avg(adr("array"),sizeof("array"));
because this function works with pointers its very time efficient and it needs no extra memory.

*)

stop := SHR(size,2)-1;
FOR i := 0 TO stop DO
	IF pt^[i] <> 0.0 THEN
		ARRAY_HAV := ARRAY_HAV + 1.0 / pt^[i];
	ELSE
		ARRAY_HAV := 0.0;
		RETURN;
	END_IF;
END_FOR;
ARRAY_HAV := UINT_TO_REAL(stop + 1) / ARRAY_HAV;


(* revision history
hm	2. apr 2008	rev 1.0
	original version

hm	10. mar. 2009	rev 1.1
	real constants updated to new systax using dot

*)

END_FUNCTION

// POUs/Mathematical/Array/ARRAY_MAX
FUNCTION ARRAY_MAX : REAL
VAR_INPUT
	pt : POINTER TO ARRAY[0..32000] OF REAL;
	size : UINT;
END_VAR
VAR
	i: UINT;
	stop: UINT;
END_VAR

(*
version 1.1	16. mar. 2008
programmer 	hugo
tested by		tobias

this function will calculate the max value of a given array.
the function needs to be called:	array_max(adr("array"),sizeof("array"));
because this function works with pointers its very time efficient and it needs no extra memory.

*)

stop := (size -SIZEOF(pt)) / SIZEOF(pt);
array_max := pt^[0];
FOR i := 1 TO stop DO
	IF pt^[i] > array_max THEN array_max := pt^[i]; END_IF;
END_FOR;

(* revision history
hm	2. oct 2006		rev 1.0
	original version

hm	16. mar. 2008	rev 1.1
	changed input size to uint
*)

END_FUNCTION

// POUs/Mathematical/Array/ARRAY_MIN
FUNCTION ARRAY_MIN : REAL
VAR_INPUT
	pt : POINTER TO ARRAY[0..32000] OF REAL;
	size : UINT;
END_VAR
VAR
	i: UINT;
	stop: UINT;
END_VAR

(*
version 1.1	16. mar. 2008
programmer 	hugo
tested by		tobias

this function will calculate the min value of a given array.
the function needs to be called:	array_min(adr("array"),sizeof("array"));
because this function works with pointers its very time efficient and it needs no extra memory.

*)

stop := (size - SIZEOF(pt)) / SIZEOF(pt);
array_min := pt^[0];
FOR i := 1 TO stop DO
	IF pt^[i] < array_min THEN array_min := pt^[i]; END_IF;
END_FOR;


(* revision history
hm		2. oct. 2006
	original version

hm		16. mar. 2008
	changed type of input size to uint

*)

END_FUNCTION

// POUs/Mathematical/Array/ARRAY_SDV
FUNCTION ARRAY_SDV : REAL
VAR_INPUT
	pt : POINTER TO ARRAY[0..32000] OF REAL;
	size : UINT;
END_VAR


(*
version 1.1	16. mar 2008
programmer 	hugo
tested by		tobias

this function will calculate the standard deviation of a given array.
the function needs to be called:	array_sdv(adr("array"),sizeof("array"));
because this function works with pointers its very time efficient and it needs no extra memory.

*)

(* standard deviation is simply the square root of the variance *)

array_sdv := SQRT(array_var(pt, size));

(* revision history
hm 	1.4.2007		rev 1.0
	function created

hm	16. mar. 2008	rev 1.1
	changed type of input size to uint

*)

END_FUNCTION

// POUs/Mathematical/Array/ARRAY_VAR
FUNCTION ARRAY_VAR : REAL
VAR_INPUT
	pt : POINTER TO ARRAY[0..32000] OF REAL;
	size : UINT;
END_VAR
VAR
	avg : REAL;
	i: UINT;
	stop: UINT;
END_VAR

(*
version 1.3	10. mar. 2009
programmer 	hugo
tested by		tobias

this function will calculate the variance of a given array.
the function needs to be called:	array_var(adr("array"),sizeof("array"));
because this function works with pointers its very time efficient and it needs no extra memory.

*)

(* at first we calualte the arithmetic average of the array *)

stop := SHR(size,2)-1;
avg := pt^[0];
FOR i := 1 TO stop DO
	avg := avg + pt^[i];
END_FOR;
avg := avg / UINT_TO_REAL(stop + 1);

(* in a second run we calculate the variance of the array *)

array_var := (pt^[0] - avg) * (pt^[0] - avg);
FOR i := 1 TO stop DO
	array_var := array_var + (pt^[i] - avg) * (pt^[i] - avg);
END_FOR;
ARRAY_VAR := ARRAY_VAR / UINT_TO_REAL(stop);

(* revision history
hm 	1.4.2007	rev 1.0
	function created

hm	12.12.2007	rev 1.1
	changed code for better performance

hm	16. mar. 2008	rev 1.2
	changed type of input size to uint

hm	10. mar. 2009	rev 1.3
	added type conversions for compatibility reasons
*)

END_FUNCTION

// POUs/Mathematical/Array/ARRAY_SPR
FUNCTION ARRAY_SPR : REAL
VAR_INPUT
	pt : POINTER TO ARRAY[0..32000] OF REAL;
	size : UINT;
END_VAR
VAR
	i: UINT;
	stop: UINT;
	array_max : REAL;
	array_min : REAL;
END_VAR

(*
version 1.1	16. mar. 2008
programmer 	hugo
tested by		tobias

this function will calculate the spread of a given array.
the function needs to be called:	array_spr(adr("array"),sizeof("array"));
for example: spread of [12,0,4,1,7] is 12 - 0 = 12.
because this function works with pointers its very time efficient and it needs no extra memory.

*)

stop := (size -SIZEOF(pt)) / SIZEOF(pt);
array_min := pt^[0];
array_max := pt^[0];
FOR i := 1 TO stop DO
	IF pt^[i] > array_max THEN array_max := pt^[i];
	ELSIF pt^[i] < array_min THEN array_min := pt^[i];
	END_IF;
END_FOR;
array_spr := array_max - array_min;


(* revision history
hm 	2. oct. 2006	rev 1.0
	original version

hm	16. mar. 2008	rev 1.1
	changed type of input size to uint

*)

END_FUNCTION

// POUs/Mathematical/Array/ARRAY_SUM
FUNCTION ARRAY_SUM : REAL
VAR_INPUT
	pt : POINTER TO ARRAY[0..32000] OF REAL;
	size : UINT;
END_VAR
VAR
	i: UINT;
	stop: UINT;
END_VAR


(*
version 1.1	16. mar. 2008
programmer 	hugo
tested by		tobias

this function will calculate the sum of a given array.
the function needs to be called:	array_sum(adr("array"),sizeof("array"));
because this function works with pointers its very time efficient and it needs no extra memory.

*)

stop := (size -SIZEOF(pt)) / SIZEOF(pt);
array_sum := pt^[0];
FOR i := 1 TO stop DO
	array_sum := array_sum + pt^[i];
END_FOR;

(* revision history
hm 	2. oct. 2006	rev 1.0
	function created

hm	16. mar. 2008	rev 1.1
	changed type of input size to uint

*)

END_FUNCTION

// POUs/Mathematical/Array/ARRAY_TREND
FUNCTION ARRAY_TREND : REAL
VAR_INPUT
	pt : POINTER TO ARRAY[0..32000] OF REAL;
	size : UINT;
END_VAR
VAR
	i: UINT;
	stop: UINT;
	x: REAL;
	stop2: UINT;
END_VAR

(*
version 1.3	10. mar. 2009
programmer 	hugo
tested by		tobias

this function will calculate the trend of a given array.
trend will calculate the avg of the first half of the array and then the avg of the second half, trend = avg2 - avg1.
for example:  [0,1,4,5,3,4,6,3] = 4 - 2.5 = 1.5
the function needs to be called:	array_trend(adr("array"),sizeof("array"));
because this function works with pointers its very time efficient and it needs no extra memory.

*)

stop := SHR(size,2)-1;
stop2 := SHR(stop,1);
FOR i := 0 TO stop2 DO x := x - pt^[i]; END_FOR;
IF EVEN(UINT_TO_INT(stop)) THEN
	FOR i := stop2 TO stop DO X := X + pt^[i]; END_FOR;
ELSE
	FOR i := stop2 + 1 TO stop DO X := X + pt^[i]; END_FOR;
END_IF;
ARRAY_TREND := x / UINT_TO_REAL(stop2 + 1);

(* revision history
hm	2 oct 2007	rev 1.0
	original version

hm	12 dec 2007	rev 1.1
	changed code for better performance

hm	16. mar. 2008	rev 1.2
	changed type of input size to uint

hm	10. mar. 2009	rev 1.3
	added type conversions for compatibility reasons
*)

END_FUNCTION

// POUs/Mathematical/ASINH
FUNCTION ASINH : REAL
VAR_INPUT
	X : REAL;
END_VAR


(*
version 1.3	10. mar 2009
programmer 	hugo
tested by		tobias

this function calculates the arcus sin hyperbolicus

*)

ASINH := LN(SQRT(X * X + 1.0)+X);

(* revision history
hm		12 jan 2007	rev 1.0
	original version

hm		2. dec 2007	rev 1.1
	changed code for better performance

hm		16.3. 2007		rev 1.2
	changed sequence of calculations to improve performance

hm	10. mar. 2009		rev 1.3
	real constants updated to new systax using dot

*)

END_FUNCTION

// POUs/Engineering/conversion/ASTRO
FUNCTION_BLOCK ASTRO
VAR_INPUT
	m : REAL;
	AE : REAL;
	PC : REAL;
	LJ : REAL;
END_VAR
VAR_OUTPUT
	Ym : REAL;
	YAE : REAL;
	YPC : REAL;
	YLJ : REAL;
END_VAR


(*
version 1.1	11. mar. 2009
programmer 	hugo
tested by		oscat

this function converts different length units
any unused input can simply be left open.
different inputs connected at the same time will be added up.

*)

YAE :=	AE
		+ m * 6.6845871535E-012
		+ PC * 206265.0
		+ LJ * 63240.0;
Ym := YAE * 149.597870E9;
YPC := YAE * 4.8481322570E-006;
YLJ := YAE * 1.5812776724E-005;


(*
Länge Meter m SI-Basiseinheit
Astronomische Einheit* AE 1 AE = 149,597 870 · E9 m
Parsec pc 1 pc = 206265 AE = 30,857 · E15 m
Lichtjahr Lj 1 Lj = 9,460 530 · E15 m = 63240 AE = 0,306 59 pc
Ångström Å 1 Å = El0 m
typograph. Punkt p 1 p = 0,376 065 mm  im Druckereigewerbe
inch** in 1 in = 2,54 · E2 m = 25,4 mm***
foot ft 1 ft = 0,3048 m = 30,48 cm
yard yd 1 yd = 0,9144 m
mile mile 1 mile = 1609,344 m
Internat. Seemeile sm 1 sm = 1852 m
Fathom fm 1 fm = 1,829 m  in der Seeschifffahrt
*)

(* revision history

hm	27. mar. 2007	rev 1.0
	original version

hm	11. mar. 2009	rev 1.1
	improved code

*)

END_FUNCTION_BLOCK

// POUs/Engineering/conversion/LENGTH
FUNCTION_BLOCK LENGTH
VAR_INPUT
	m : REAL;
	p : REAL;
	in : REAL;
	ft : REAL;
	yd : REAL;
	mile : REAL;
	sm : REAL;
	fm : REAL;
END_VAR
VAR_OUTPUT
	Ym : REAL;
	Yp : REAL;
	Yin : REAL;
	Yft : REAL;
	Yyd : REAL;
	Ymile : REAL;
	Ysm : REAL;
	Yfm : REAL;
END_VAR


(*
version 1.1	11. mar. 2009
programmer 	hugo
tested by		oscat

this function converts different length units
any unused input can simply be left open.
different inputs connected at the same time will be added up.

*)

Ym :=	m
		+ p * 0.000376065
		+ in * 0.0254
		+ ft * 0.3048
		+ yd * 0.9144
		+ mile * 1609.344
		+ sm * 1852.0
		+ fm * 1.829;
Yp := Ym * 2659.11478068951;
Yin := Ym * 39.37007874016;
Yft := Ym * 3.28083989501;
Yyd := Ym * 1.09361329834;
Ymile := Ym * 0.00062137119;
Ysm := Ym * 0.00053995680;
Yfm := Ym * 0.54674685621;

(*
Länge Meter m SI-Basiseinheit
Astronomische Einheit* AE 1 AE = 149,597 870 · E9 m
Parsec pc 1 pc = 206265 AE = 30,857 · E15 m
Lichtjahr Lj 1 Lj = 9,460 530 · E15 m = 63240 AE = 0,306 59 pc
Ångström Å 1 Å = El0 m
typograph. Punkt p 1 p = 0,376 065 mm  im Druckereigewerbe
inch** in 1 in = 2,54 · E2 m = 25,4 mm***
foot ft 1 ft = 0,3048 m = 30,48 cm
yard yd 1 yd = 0,9144 m
mile mile 1 mile = 1609,344 m
Internat. Seemeile sm 1 sm = 1852 m
Fathom fm 1 fm = 1,829 m  in der Seeschifffahrt
*)

(* revision history

hm	27. mar. 2007	rev 1.0
	original version

hm	11. mar. 2009	rev 1.1
	improved code

*)

END_FUNCTION_BLOCK

// POUs/Mathematical/ATAN2
FUNCTION ATAN2 : REAL
VAR_INPUT
	Y : REAL;
	X : REAL;
END_VAR


(*
version 1.2	10. mar. 2009
programmer 	hugo
tested by		oscat

this function calculates the angle in a coordinate system in rad.

*)

IF X > 0.0 THEN
	ATAN2 := ATAN(Y/X);
ELSIF X < 0.0 THEN
	IF Y >=0.0 THEN
		ATAN2 := ATAN(Y/X) + MATH.PI;
	ELSE
		ATAN2 := ATAN(Y/X) - MATH.PI;
	END_IF;
ELSIF Y > 0.0 THEN
	ATAN2 := MATH.PI05;
ELSIF Y < 0.0 THEN
	ATAN2 := -MATH.PI05;
ELSE
	ATAN2 := 0.0;
END_IF;


(* revision history
hm	20.  apr. 2008	rev 1.0
	original version

hm	18. oct. 2008	rev 1.1
	changed to use math constants

hm	10. mar. 2009	rev 1.2
	real constants updated to new systax using dot

*)

END_FUNCTION

// POUs/Mathematical/ATANH
FUNCTION ATANH : REAL
VAR_INPUT
	X : REAL;
END_VAR


(*
version 1.2	10. mar. 2009
programmer 	hugo
tested by		tobias

this function calculates the arcus tangens hyperbolicus

*)

ATANH := LN((1.0 + x)/(1.0 - x)) * 0.5;


(* revision history
hm		12 jan 2007	rev 1.0
	original version

hm		5. jan 2008	rev 1.1
	improved code for better performance

hm	10. mar. 2009		rev 1.2
	real constants updated to new systax using dot

*)

END_FUNCTION

// POUs/Logic/generators/B_TRIG
FUNCTION_BLOCK B_TRIG
VAR_INPUT
	CLK : BOOL;
END_VAR
VAR_OUTPUT
	Q : BOOL;
END_VAR
VAR
	edge : BOOL;
END_VAR

(*
version 1.0	4. aug. 2006
programmer 	hugo
tested by		tobias

this block is similar to R_trig and F_trig but it generates a pulse on rising and falling edge.

*)

Q := clk XOR edge;
edge := CLK;


(* revision history
hm		4. aug. 2006	rev 1.0
	original version

*)

END_FUNCTION_BLOCK

// POUs/Engineering/measurements/BAR_GRAPH
FUNCTION_BLOCK BAR_GRAPH
VAR_INPUT
	X : REAL;
	rst : BOOL;
END_VAR
VAR_INPUT CONSTANT
	trigger_Low : REAL;
	trigger_High : REAL;
	Alarm_low : BOOL;
	Alarm_high : BOOL;
	log_scale : BOOL;
END_VAR
VAR_OUTPUT
	LOW, Q1, Q2, Q3, Q4, Q5, Q6, HIGH : BOOL;
	Alarm : BOOL;
	Status : BYTE;
END_VAR
VAR
	init : BOOL;
	T1, T2, T3, T4, T5 : REAL;
END_VAR
VAR
	temp : REAL;
END_VAR

(*
	version 1.2	6 jan 2008
	programmer 	hugo
	tested BY	hans

bar graph is a muti window comparator which displays an analog input signal on 8 digital outputs.
only one output is active a any given time depending on the value of the input signal.
the output can be of linear or logarithmic scale.

*)

IF NOT init THEN
	init := TRUE;
	IF log_scale THEN
		temp := EXP(LN(Trigger_high / Trigger_low) * 0.166666666666666666666);
		T1 := trigger_low * temp;
		T2 := T1 * temp;
		T3 := T2 * temp;
		T4 := T3 * temp;
		T5 := T4 * temp;
	ELSE
		temp := (trigger_high - trigger_low) * 0.142857142;
		T1 := trigger_low + temp;
		T2 := T1 + temp;
		T3 := T2 + temp;
		T4 := T3 + temp;
		T5 := T4 + temp;
	END_IF;
END_IF;

(* clear outputs before checking *)
Q1 := FALSE;
Q2 := FALSE;
Q3 := FALSE;
Q4 := FALSE;
Q5 := FALSE;
Q6 := FALSE;
status := 110;

(* low, high and alarm can only be cleared with rst depending on alarm_low and alarm_high *)
IF NOT alarm_low THEN low := FALSE; END_IF;
IF NOT alarm_high THEN high := FALSE; END_IF;
IF rst THEN
	alarm := FALSE;
	low := FALSE;
	high := FALSE;
END_IF;

(* check and set outputs *)
IF X < trigger_low THEN
	Low := TRUE;
	status := 111;
	IF alarm_low THEN
		alarm := TRUE;
		status := 1;
	END_IF;
ELSIF X < T1 THEN
	Q1 := TRUE;
ELSIF x < t2 THEN
	Q2 := TRUE;
ELSIF x < t3 THEN
	Q3 := TRUE;
ELSIF x < T4 THEN
	Q4 := TRUE;
ELSIF x < T5 THEN
	q5 := TRUE;
ELSIF x < trigger_high THEN
	q6 := TRUE;
ELSE
	high := TRUE;
	status := 112;
	IF alarm_high THEN
		alarm := TRUE;
		status := 2;
	END_IF;
END_IF;

(* revision history
hm	22. feb 2007	rev 1.0
	original version

hm	2. dec 2007		rev 1.1
	chaged code for better performance

hm	6. jan 2008		rev 1.2
	further performance improvement

*)

END_FUNCTION_BLOCK

// POUs/Mathematical/WINDOW
FUNCTION WINDOW : BOOL
VAR_INPUT
	low : REAL;
	in : REAL;
	high : REAL;
END_VAR


(*
	version 1.1	22 jan 2007
	programmer 	hugo
	tested BY	tobias

this checks a signal if the signal is between the upper and lower limit
*)

WINDOW := in < high AND in > low;


(* revision history
hm	22.1.2007	rev 1.1
	changed the order of inputs to low, in, high

*)

END_FUNCTION

// POUs/Logic/gate logic/BCDC_TO_INT
FUNCTION BCDC_TO_INT : INT
VAR_INPUT
	IN : BYTE;
END_VAR


(*
version 1.1 30. jun. 2008
programmer 	hugo
tested by	oscat

this function converts a two digit bcd number into an integer.

*)

BCDC_TO_INT := (in AND 16#0F) + (SHR(in,4) * 10);

(* revision history
hm	13.12.2007	rev 1.0
	original version

hm	30.6.2008	rev 1.1
	changed name BCD_TO_INT to BCDC_TO_INT to avoid collision with util.lib

*)

END_FUNCTION

// POUs/Mathematical/BETA
FUNCTION BETA : REAL
VAR_INPUT
	X : REAL;
	Y : REAL;
END_VAR


(*
version 1.0	26. oct. 2008
programmer 	hugo
tested by		oscat

this function calculates the beta function for real number > 0.

*)

BETA := GAMMA(X) * GAMMA(Y) / GAMMA(x + y);


(* revision history
hm	26. oct. 2008	rev 1.0
	original version

*)

END_FUNCTION

// POUs/Mathematical/GAMMA
FUNCTION GAMMA : REAL
VAR_INPUT
	X : REAL;
END_VAR


(*
version 1.3	10. mar. 2009
programmer 	hugo
tested by		oscat

this function calculates the stirling function which is an approximation for the gamma function

*)

IF x > 0.0 THEN
	GAMMA := SQRT(math.PI2 / X) * EXPT(math.E_INV * (x + 1.0 / (12.0 * x - 0.1 / X)), X);
END_IF;


(* the stirling formula is not very accurate for small values of X
IF X >=0 THEN GAMMA := SQRT(math.PI2 * X) * EXPT(X / math.E, X); END_IF;
*)





(* revision history
hm	10.12.2007	rev 1.0
	original version

hm	18. oct. 2008	rev 1.1
	using math constants

hm	26. oct. 2008	rev 1.2
	using new formula with better accuracy

hm	10. mar. 2009	rev 1.3
	real constants updated to new systax using dot

*)

END_FUNCTION

// POUs/Engineering/conversion/BFT_TO_MS
FUNCTION BFT_TO_MS : REAL
VAR_INPUT
	BFT : INT;
END_VAR


(*
version 1.0	12. jun 2008
programmer 	hugo
tested by		oscdat

this function converts wind speed from beaufort to m/s
*)

BFT_TO_MS := EXPT(BFT, 1.5) * 0.836;


(* revision history
hm	12. 6. 2008		rev 1.0
	original version

*)

END_FUNCTION

// POUs/String/BIN_TO_BYTE
FUNCTION BIN_TO_BYTE : BYTE
VAR_INPUT
	BIN : STRING(12);
END_VAR
VAR
	pt : POINTER TO BYTE;
	i: INT;
	X: BYTE;
	stop: INT;
END_VAR

(*
version 1.2	26. jul 2009
programmer 	hugo
tested by		oscat

BINARY_TO_byte converts a binary string into a byte.

*)

pt := ADR(bin);
stop := LEN(bin);
FOR I := 1 TO stop DO
	x := pt^;
	(* calculate the value of the digit *)
	IF X = 48 THEN
		BIN_TO_BYTE := SHL(BIN_TO_BYTE,1);
	ELSIF X = 49 THEN
		BIN_TO_BYTE := SHL(BIN_TO_BYTE,1) OR 1;
	END_IF;
	pt := pt + 1;
END_FOR;



(* revision histroy
hm	18. jun. 2008	rev 1.0
	original release

hm	20. sep. 2008	rev 1.1
	changed length of input string from 20 to 12

hm	26. jul. 2009	rev 1.2
	optimized code
*)

END_FUNCTION

// POUs/String/BIN_TO_DWORD
FUNCTION BIN_TO_DWORD : DWORD
VAR_INPUT
	BIN : STRING(40);
END_VAR
VAR
	pt : POINTER TO BYTE;
	i: INT;
	X: BYTE;
	stop: INT;
END_VAR

(*
version 1.2	26. jul. 2009
programmer 	hugo
tested by		oscat

BINARY_TO_DWORD converts a binary string into a dword.

*)

pt := ADR(bin);
stop := LEN(bin);
FOR I := 1 TO stop DO
	x := pt^;
	(* calculate the value of the digit *)
	IF X = 48 THEN
		BIN_TO_DWORD := SHL(BIN_TO_DWORD,1);
	ELSIF X = 49 THEN
		BIN_TO_DWORD := SHL(BIN_TO_DWORD,1) OR 1;
	END_IF;
	pt := pt + 1;
END_FOR;



(* revision histroy
hm	18. jun. 2008	rev 1.0
	original release

hm	20. sep. 2008	rev 1.1
	changed length of input dtring from 20 to 40

hm	26. jul 2009	rev 1.2
	optimized code
*)

END_FUNCTION

// POUs/Mathematical/BINOM
FUNCTION BINOM : DINT
VAR_INPUT
	N : INT;
	K : INT;
END_VAR

VAR
	i: INT;
END_VAR


(*
version 1.0	25. oct. 2008
programmer 	hugo
tested by		tobias

this function calculates the binomialkoefficient (N over k)

*)

IF 2 * K > n THEN
	k := n - k;
END_IF;
IF k > n THEN
	RETURN;
ELSIF k = 0 OR k = n THEN
	BINOM := 1;
ELSIF k = 1 THEN
	BINOM := n;
ELSE
	BINOM := n;
	n := n + 1;
	FOR i := 2 TO k DO
		BINOM := BINOM * (n - i) / i;
	END_FOR;
END_IF;



(*
binomialkoeffizient(n, k)
1  wenn k = 0 return 1
2  wenn 2k > n
3      dann führe aus ergebnis \leftarrow binomialkoeffizient(n, n-k)
4  sonst führe aus ergebnis \leftarrow n
5          von i \leftarrow 2 bis k
6              führe aus ergebnis \leftarrow ergebnis \cdot (n + 1 - i)
7                        ergebnis \leftarrow ergebnis : i
8  return ergebnis
*)



(* revision history
hm	25. oct. 2008	rev 1.0
	original version


*)

END_FUNCTION

// POUs/Logic/gate logic/BIT_LOAD_B
FUNCTION BIT_LOAD_B : BYTE
VAR_INPUT
	IN : BYTE;
	VAL : BOOL;
	POS : INT;
END_VAR
VAR CONSTANT
	dat : BYTE := 1;
END_VAR

(*
version 1.1	16. mar 2008
programmer 	hugo
tested by	tobias

this function loads a bit into a byte at position pos.
 *)

IF VAL THEN
	BIT_LOAD_B := in OR SHL(dat,pos);
ELSE
	BIT_LOAD_B := in AND (NOT SHL(dat,pos));
END_IF;


(* revision history
hm	29. feb 2008	rev 1.0
	original version

hm	16. mar 2008	rev 1.1
	change input bit to val for compatibility reasons
*)

END_FUNCTION

// POUs/Logic/gate logic/BIT_LOAD_B2
FUNCTION BIT_LOAD_B2 : BYTE
VAR_INPUT
	I : BYTE;
	D : BOOL;
	P : INT;
	N : INT;
END_VAR


(*
version 1.0 18. oct. 2008
programmer 	hugo
tested by	tobias

this function loads N bits of D at pos P in Byte I

*)

IF D THEN
	BIT_LOAD_B2 := ROL(SHR(BYTE#255, 8 - N) OR ROR(i, P), P);
ELSE
	BIT_LOAD_B2 := ROL(SHL(BYTE#255, N) AND ROR(I, P), P);
END_IF;



(* revision history
hm	18. oct. 2008	rev 1.0
	original version


*)

END_FUNCTION

// POUs/Logic/gate logic/BIT_LOAD_DW
FUNCTION BIT_LOAD_DW : DWORD
VAR_INPUT
	IN : DWORD;
	VAL : BOOL;
	POS : INT;
END_VAR
VAR CONSTANT
	dat : DWORD := 1;
END_VAR

(*
version 1.1	16. mar 2008
programmer 	hugo
tested by	tobias

this function loads a bit into a DWord at position pos.
 *)

IF val THEN
	BIT_LOAD_DW := in OR SHL(dat,pos);
ELSE
	BIT_LOAD_DW := in AND (NOT SHL(dat,pos));
END_IF;


(* revision history
hm	29. feb 2008	rev 1.0
	original version

hm	16. mar 2008	rev 1.1
	change input bit to val for compatibility reasons
*)

END_FUNCTION

// POUs/Logic/gate logic/BIT_LOAD_DW2
FUNCTION BIT_LOAD_DW2 : DWORD
VAR_INPUT
	I : DWORD;
	D : BOOL;
	P : INT;
	N : INT;
END_VAR


(*
version 1.0 18. oct. 2008
programmer 	hugo
tested by	tobias

this function loads N bits of D at pos P in DWORD I

*)

IF D THEN
	BIT_LOAD_DW2 := ROL(SHR(DWORD#4294967295, 32 - N) OR ROR(i, P), P);
ELSE
	BIT_LOAD_DW2 := ROL(SHL(DWORD#4294967295, N) AND ROR(I, P), P);
END_IF;



(* revision history
hm	18. oct. 2008	rev 1.0
	original version


*)

END_FUNCTION

// POUs/Logic/gate logic/BIT_LOAD_W
FUNCTION BIT_LOAD_W : WORD
VAR_INPUT
	IN : WORD;
	VAL : BOOL;
	POS : INT;
END_VAR
VAR CONSTANT
	dat : WORD := 1;
END_VAR

(*
version 1.1	16. mar 2008
programmer 	hugo
tested by	tobias

this function loads a bit into a Word at position pos.
 *)

IF val THEN
	BIT_LOAD_W := in OR SHL(dat,pos);
ELSE
	BIT_LOAD_W := in AND (NOT SHL(dat,pos));
END_IF;


(* revision history
hm	29. feb 2008	rev 1.0
	original version

hm	16. mar 2008	rev 1.1
	change input bit to val for compatibility reasons
*)

END_FUNCTION

// POUs/Logic/gate logic/BIT_LOAD_W2
FUNCTION BIT_LOAD_W2 : WORD
VAR_INPUT
	I : WORD;
	D : BOOL;
	P : INT;
	N : INT;
END_VAR


(*
version 1.0 18. oct. 2008
programmer 	hugo
tested by	tobias

this function loads N bits of D at pos P in WORD I

*)

IF D THEN
	BIT_LOAD_W2 := ROL(SHR(WORD#65535, 16 - N) OR ROR(i, P), P);
ELSE
	BIT_LOAD_W2 := ROL(SHL(WORD#65535, N) AND ROR(I, P), P);
END_IF;



(* revision history
hm	18. oct. 2008	rev 1.0
	original version


*)

END_FUNCTION

// POUs/Logic/gate logic/BIT_OF_DWORD
FUNCTION BIT_OF_DWORD : BOOL
VAR_INPUT
	in : DWORD;
	N : INT;
END_VAR


(*
version 1.2	6. jun. 2008
programmer 	hugo
tested by	tobias

this function extracts a single bit from the nth position from right (right is lowest bit)
the lowest Bit (Bit0 from in) is selected with N=0.
 *)

BIT_OF_DWORD := (SHR(in,N) AND 16#00000001) > 0;


(* old code used before rev 1.1
temp := SHR(in,n);
Bit_of_Dword := temp.0;
*)


(* revision history
hm	4. aug. 2006	rev 1.0
	original version

hm	29. feb 2008	rev 1.1
	improved performance

hm	6. jun. 2008	rev 1.2
	changes type of input N from byte to int
*)

END_FUNCTION

// POUs/Logic/gate logic/BIT_TOGGLE_B
FUNCTION BIT_TOGGLE_B : BYTE
VAR_INPUT
	IN : BYTE;
	POS : INT;
END_VAR


(*
version 1.0 18. oct. 2008
programmer 	hugo
tested by	tobias

this function toggles a bit of a BYTE at position pos.

*)

BIT_TOGGLE_B := SHL(BYTE#1, POS) XOR IN;




(* revision history
hm	18. oct. 2008	rev 1.0
	original version


*)

END_FUNCTION

// POUs/Logic/gate logic/BIT_TOGGLE_DW
FUNCTION BIT_TOGGLE_DW : DWORD
VAR_INPUT
	IN : DWORD;
	POS : INT;
END_VAR


(*
version 1.0 18. oct. 2008
programmer 	hugo
tested by	tobias

this function toggles a bit of a WORD at position pos.

*)

BIT_TOGGLE_DW := SHL(DWORD#1, POS) XOR IN;



(* revision history
hm	18. oct. 2008	rev 1.0
	original version


*)

END_FUNCTION

// POUs/Logic/gate logic/BIT_TOGGLE_W
FUNCTION BIT_TOGGLE_W : WORD
VAR_INPUT
	IN : WORD;
	POS : INT;
END_VAR


(*
version 1.0 18. oct. 2008
programmer 	hugo
tested by	tobias

this function toggles a bit of a WORD at position pos.

*)

BIT_TOGGLE_W := SHL(WORD#1, POS) XOR IN;



(* revision history
hm	18. oct. 2008	rev 1.0
	original version


*)

END_FUNCTION

// POUs/Building/Jalousie/BLIND_ACTUATOR
 FUNCTION_BLOCK BLIND_ACTUATOR
VAR_INPUT
	UP, DN : BOOL;
	S_IN : BYTE;
	T_UD : TIME := T#10s;
	T_ANGLE : TIME := T#3s;
END_VAR
VAR_INPUT CONSTANT
	T_LOCKOUT : TIME := t#100ms;
END_VAR
VAR_OUTPUT
	POS, ANG : BYTE;
	QU, QD : BOOL;
	STATUS : BYTE;
END_VAR
VAR
	position, angle : RMP_B;
	lock : INTERLOCK;
END_VAR

(*
version 1.3	27. jul. 2009
programmer 	hugo
tested by		oscat

blind actuator drives the up and down motor of a blind. T_lockout specifies the time between up or dn becomes active. 
To change direction there must be a minimum wait time to allow the motors to come to rest first.
the up and down outputs QU and QD are controlled by the inputs UP and DN.
the outputs pos and ang simulate the position of the blind pos = 0 means blind is down and pos = 255 = blind is up.
the angle 0 means vertical posisition of the slates and 255 means horizontal position of the slates.


*)

(* make sure only one motor is active at a given time *)
lock(i1 := UP, I2 := DN, TL := T_lockout);

(* ramp up or down to simulate the angle position of the blind slats *)
angle(e := lock.Q1 OR lock.Q2, UP := lock.Q1, PT := T_Angle);
position(e := lock.Q1 AND angle.high OR lock.Q2 AND angle.low, up := lock.Q1, PT := T_UD);

(* set the outputs *)
pos := position.Out;
ang := angle.Out;
QU := lock.Q1;
QD := lock.Q2;

(* set the status output *)
IF UP AND DN THEN
	 status := 1;			(* error up and down together are not allowed *)
ELSIF UP THEN
	status := 121;
ELSIF DN THEN
	status := 122;
ELSE
	status := S_IN;
END_IF;


(* revision history
hm	29. sep 2007	rev 1.0
	original release

hm	6. oct 2007	rev 1.1
	rearanged outputs

hm	18. oct. 2008	rev 1.2
	changed calls for rmp_B because of change in RMP_B

hm	27. jul. 2009	rev 1.3
	changes status to be 12X
*)

END_FUNCTION_BLOCK

// POUs/Engineering/signal generators/RMP_B
FUNCTION_BLOCK RMP_B
VAR_INPUT
	SET : BOOL;
	PT : TIME;
	E : BOOL := TRUE;
	UP : BOOL := TRUE;
	RST : BOOL;
END_VAR
VAR_OUTPUT
	OUT : BYTE;
	BUSY: BOOL;
	HIGH : BOOL;
	LOW : BOOL;
END_VAR
VAR
	rmp : _RMP_B;
END_VAR


(*
version 2.0	23. oct. 2008
programmer 	oscat
tested BY	oscat

this ramp generator generates a byte wide ramp with 255 steps
the generator has an asynchronous set and reset
the ramp is controlled by PT which is the total ramp time for a full sweep from 0..255
an UD input controlls the direction Up or Down and the E input enables the ramp generation
a busy output indicates that the ramp is running, busy false means output is stable.
the outputs low and high will be true when the output has reached its max or min value.

*)

(* generate ramp *)
rmp(dir := UP, E := E, TR := PT, rmp := out);

(* set or reset operation *)
IF RST THEN
	out := 0;
ELSIF SET THEN
	out := 255;
END_IF;

(* checks for outputs stable and reset or set busy flag *)
low := out = 0;
high := out = 255;
busy := NOT (low OR high) AND E;


(* revision history

hm 5.10.2006	rev 1.1
	added busy output
hm 17.1.2007	rev 1.2
	renamed input ud to up for better usability
	deleted unused variable step

hm	17.9.2007		rev 1.3
	replaced time() with t_plc_ms() for compatibility reasons

hm	28. sep 2007	rev 1.4
	added outputs on and off
	busy is now disabled while en is false
	new coding for higher accuracy and performance

hm	5. oct 2007	rev 1.5
	added statements to allow for PT to be t#0s output jumps to max or min immediately

hm	25. dec 2007	rev 1.6
	improved code for better performance

hm	16. oct. 2008	rev 1.7
	improved code for better performance

hm	18. oct. 2008	rev 1.8
	added type conversion to avoid warnings
	changed input en to e for compatibility reasons

hm	23. oct. 2008	REV 	2.0
	new code using _RMP_B

*)

END_FUNCTION_BLOCK

// POUs/Engineering/automation/INTERLOCK
FUNCTION_BLOCK INTERLOCK
VAR_INPUT
	I1, I2 : BOOL;
	TL : TIME;
END_VAR
VAR_OUTPUT
	Q1, Q2 : BOOL;
END_VAR
VAR
	T1, T2 : TOF;
END_VAR

(*
version 1.0	28 sep 2007
programmer 	hugo
tested by		tobias

INTERLOCK has two inputs I1 and I2 which drive the corresponding outputs Q1 and Q2.
the inputs signals lock each other out and therfore I1 can only drive Q1 when I2 is Low and vice versa.
The input TL specifies a dead time between two outputs can become active.
an output can only become active when the other output was not active for the time TL.

*)

(* the input signal have a run delay to lockout the other input *)
T1(IN := I1, PT := TL);
T2(IN := I2, PT := TL);

Q1 := I1 AND NOT t2.Q;
Q2 := I2 AND NOT t1.Q;


(* revision history

hm	28 sep 2007		rev 1.0
	original version

*)

END_FUNCTION_BLOCK

// POUs/Engineering/signal processing/DELAY
FUNCTION_BLOCK DELAY
VAR_INPUT
	IN : REAL;
	N : INT;
	RST : BOOL;
END_VAR
VAR_OUTPUT
	OUT : REAL;
END_VAR
VAR
	buf : ARRAY[0..31] OF REAL;
	i : INT;
	init: BOOL;
	stop: INT;
END_VAR

(*
version 1.5	23. mar. 2009
programmer 	hugo
tested by		oscat

this function block delays input values by each programm cycle
after N+1 cycles the in value has shifted to the out.
N can be any alue from 0 .. 32
if n = 0 the input will be present on the output without a delay.
f N > 32 then the output will be delayed by 32 cycles.
any high on rst will load the buffer with in.

*)

stop := LIMIT(0,N,32) - 1;
IF rst OR NOT init THEN
	init := TRUE;
	FOR i := 0 TO stop DO buf[i] := in; END_FOR;
	out := in;
	i := 0;
ELSIF stop < 0 THEN
	out := in;
ELSE
	out := buf[i];
	buf[i] := in;
	i := INC1(i, N);
END_IF;



(* revision history
hm 1.10.2006		rev 1.1
	corrected error in buffer management

hm 19.1.2007		rev 1.2
	changed reset to load the value of in instead of 0

hm	27. oct. 2008	rev 1.3
	improved performance

hm	23. feb.2009	rev 1.4
	corrected an index problem

hm	23. mar. 2009	rev 1.5
	corrected non standard write to input N

*)

END_FUNCTION_BLOCK

// POUs/Mathematical/INC1
FUNCTION INC1 : INT
VAR_INPUT
	X : INT;
	N : INT;
END_VAR



(*
version 1.2	23. feb. 2009
programmer 	hugo
tested by	oscat

This is a increment function which increments the variable X by 1 and if N is reached, it begins with 0 instead of N again.
inc1(X,3) will generate 0,1,2,0,1,.....

*)

IF X >= N - 1 THEN
	INC1 := 0;
ELSE
	INC1 := X + 1;
END_IF;



(* revision history
hm	13. oct. 2008	rev 1.0
	original version

hm	22. oct. 2008	rev 1.1
	added statement to return value for compatibility reasons

hm	23. feb. 2009	rev 1.2
 	when inc1 is called with X >= N inc will continue with 0
*)

END_FUNCTION

// POUs/Mathematical/INC
FUNCTION INC : INT
VAR_INPUT
	X : INT;
	D : INT;
	M : INT;
END_VAR


(*
version 1.1	15. jan 2008
programmer 	hugo
tested by	oscat

This is a increment function which increments the input X by the value D and compares the result with M.
if the output exceeds M it will continue to count from 0 again.

*)

INC := (X + D + M + 1) MOD (M + 1);

(* revision history
hm	7. feb 2007		REV 1.0
	original version

hm	15. jan 2008	rev 1.1
	allow for neagtive increment

*)

END_FUNCTION

// POUs/Building/Jalousie/BLIND_CONTROL
FUNCTION_BLOCK BLIND_CONTROL
VAR_INPUT
	UP, DN : BOOL;
	S_IN : BYTE;
	PI : BYTE;
	AI : BYTE;
	T_UD, T_ANGLE : TIME;
END_VAR
VAR_INPUT CONSTANT
	SENS : BYTE := 5;
	T_LOCKOUT: TIME := T#100ms;
END_VAR
VAR_OUTPUT
	POS, ANG : BYTE;
	MU, MD : BOOL;
	STATUS : BYTE;
END_VAR
VAR
	act : BLIND_ACTUATOR;
	delta : BYTE;
END_VAR

(*
version 1.4	27. jul 2009
programmer 	hugo
tested by		tobias


*)

IF UP AND DN THEN
	(* automatic modus detected *)
	(* first find correct position *)
	IF BYTE_TO_INT(act.pos) < BYTE_TO_INT(pi) - delta THEN
		act.UP := TRUE;
		act.DN := FALSE;
		delta := 0;
		STATUS := 121;
	ELSIF BYTE_TO_INT(act.pos) > BYTE_TO_INT(pi) + delta THEN
		act.UP := FALSE;
		act.DN := TRUE;
		delta := 0;
		STATUS := 122;
	(* regulate angle *)
	ELSIF BYTE_TO_INT(act.ang) < BYTE_TO_INT(ai) - delta AND T_angle > T#100ms THEN
		act.UP := TRUE;
		act.DN := FALSE;
		delta := 0;
		STATUS := 123;
	ELSIF BYTE_TO_INT(act.ang) > BYTE_TO_INT(ai) + delta AND T_angle > T#100ms THEN
		act.UP := FALSE;
		act.DN := TRUE;
		delta := 0;
		STATUS := 124;
	(* correct position reached *)
	ELSE
		act.UP := FALSE;
		act.DN := FALSE;
		delta := sens;
		STATUS := S_IN;
	END_IF;
ELSE
	act.UP := UP;
	act.DN := DN;
	STATUS := S_IN;
END_IF;

(* blind control calls blind_actuator *)
act(T_UD:=T_UD, T_ANGLE:=T_ANGLE, T_lockout := T_Lockout);
pos := act.pos;
ang := act.ang;
MU := act.QU;
md := act.QD;
status := act.status;

(* revision history
hm	29. sep 2007	rev 1.0
	original release

hm	6. oct 2007	rev 1.1
	rearranged outputs
	integrated blind_actuator into blind_control

hm	16. oct 2007	rev 1.2
	ignore angle when t_angle = 0

hm 29. oct 2007	rev 1.3
	added lockout configuration time for motor direction change
	sens has a setup value of 5

hm	27. jul. 2009	rev 1.4
	changed status handling

*)

END_FUNCTION_BLOCK

// POUs/Building/Jalousie/BLIND_CONTROL_S
FUNCTION_BLOCK BLIND_CONTROL_S
VAR_INPUT
	UP, DN : BOOL;
	S_IN : BYTE := 125;
	PI : BYTE;
	T_UD : TIME;
	RU : BOOL;
	RD : BOOL;
END_VAR
VAR_INPUT CONSTANT
	T_LOCKOUT: TIME := T#100ms;
	T_EXT : TIME;
	EXT_TRIG : BYTE := 5;
	R_POS_TOP : BYTE := 255;
	R_POS_BOT : BYTE;
END_VAR
VAR_OUTPUT
	POS : BYTE;
	MU, MD : BOOL;
	STATUS : BYTE;
END_VAR
VAR
	rmp : _RMP_NEXT;
	tx, last : TIME;
	PI_last: BYTE;
END_VAR


(*
version 1.1	27. jul. 2009
programmer 	hugo
tested by		heinz


*)

(* status definition
	121 = manual up				manual up operation UP = true and DN = false
	122 = manual down			manual down operation DN = true and UP = false
	123 = auto positioning		automatic mode DN = UP = TRUE
	124 = revert					revert from top or bottom
	125 = nothing					default input for S_IN
	127 = Lockout time			lockout between directional change
	128 = calibrate				calibrate after power up
	129 = extend					extend runtime at top or bottom for continuous calibration
*)

(* read system time *)
tx := DWORD_TO_TIME(T_PLC_MS());

(* check inputs and start state machine *)
IF UP  AND NOT DN THEN
	(*  manual UP *)
	rmp.IN := 255;
	STATUS := 121;
ELSIF DN AND NOT UP THEN
	(* manual DN *)
	rmp.IN := 0;
	STATUS := 122;
ELSIF NOT (UP OR DN) THEN
	(* manual standby mode *)
	rmp.IN := PI;
	STATUS := S_IN;
END_IF;

(* simulate pos output *)
rmp(E := UP OR DN, TR := T_UD, TF := T_UD, TL := T_LOCKOUT, OUT := POS);

(* state machine *)
CASE STATUS OF
	0:		(* power up init *)
		last := tx;
		PI_last := PI XOR BYTE#255;
		STATUS := 128;		(* calibrate *)

	121: 	(* manual up *)
		MU := TRUE;
		MD := FALSE;
		IF POS >= (BYTE#255 - EXT_TRIG) THEN
			(* extend cycle if top is reached *)
			POS := 255;
			last := tx;
			STATUS := 129;	(* extend *)
		END_IF;

	122:	(* manual down *)
		MD := TRUE;
		MU := FALSE;
		IF POS <= EXT_TRIG THEN
			(* extend cycle if bottom is reached *)
			POS := 0;
			last := tx;
			STATUS := 129;	(* extend *)
		END_IF;

	123:	(* auto positioning *)
		MD := rmp.DN;
		MU := rmp.UP;
		IF NOT (rmp.DN OR rmp.UP) THEN
			(* automatic position is reached *)
			IF POS <= EXT_TRIG THEN
				(* extend at bottom *)
				MD := TRUE;
				last := tx;
				STATUS := 129;	(* extend *)
			ELSIF POS >= (BYTE#255 - EXT_TRIG)  THEN
				(* extend at top *)
				MU := TRUE;
				last := tx;
				STATUS := 129;	(* extend *)
			ELSE
				STATUS := S_IN;
			END_IF;
		END_IF;

	124:	(* revert from top or bottom *)
		MD := rmp.DN;
		MU := rmp.UP;
		IF NOT(rmp.DN OR rmp.UP) THEN
			PI_last := PI;
			STATUS := S_IN;
		END_IF;

	127:	(* lockout time *)
		IF (tx - last) >= T_LOCKOUT THEN
			IF POS = 0 AND RU THEN
				rmp.IN := R_POS_BOT;
				STATUS := 124;	(* revert *)
			ELSIF pos = 255 AND RD THEN
				rmp.IN := R_POS_TOP;
				STATUS := 124;	(* revert *)
			ELSE
				STATUS := S_IN;
			END_IF;
		END_IF;

	128:	(* calibration *)
		MU := TRUE;
		MD := FALSE;
		POS := 255;
		IF (tx - last) >= (T_UD +  T_EXT) THEN
			MU := FALSE;
			last := tx;
			STATUS := 127;	(* lockout *)
		END_IF;

	129: (* extend mode *)
		IF (tx - last) >= T_EXT THEN
			MU := FALSE;
			MD := FALSE;
			last := tx;
			STATUS := 127;	(* lockout *)
		END_IF;

ELSE
	MU := FALSE;
	MD := FALSE;
	IF PI <> PI_last THEN
		PI_last := PI;
		rmp.IN := PI;
		STATUS := 123;	(* auto positioning *)
	ELSE
		STATUS := S_IN;
	END_IF;
END_CASE;



(* revision history

hm	9. mar. 2009	rev 1.0
	original release

hf	27. jul 2009	rev 1.1
	major code changes and updates

*)

END_FUNCTION_BLOCK

// POUs/Building/Jalousie/BLIND_INPUT
FUNCTION_BLOCK BLIND_INPUT
VAR_INPUT
	POS, ANG : BYTE;
	S1, S2 : BOOL;
	IN : BOOL;
	PI, AI : BYTE;
END_VAR
VAR_INPUT CONSTANT
	SINGLE_SWITCH : BOOL;
	CLICK_EN : BOOL := TRUE;
	CLICK_TIME : TIME := T#500ms;
	MAX_RUNTIME : TIME := T#60s;
	MANUAL_TIMEOUT: TIME := T#1h;
	DEBOUNCE_TIME : TIME := T#20ms;
	DBL_CLK1 : BOOL := FALSE;
	DBL_POS1 : BYTE;
	DBL_ANG1 : BYTE;
	DBL_CLK2 : BOOL := FALSE;
	DBL_POS2 : BYTE := 255;
	DBL_ANG2 : BYTE := 255;
	D1_TOGGLE : BOOL := TRUE;
	D2_TOGGLE : BOOL := TRUE;
	MASTER_MODE : BOOL;
END_VAR
VAR_OUTPUT
	QU, QD : BOOL;
	STATUS : BYTE;
	PO, AO : BYTE;
	D1, D2 : BOOL;
END_VAR
VAR
	s1e, s2e : TOF;
	s1d, s2d : CLICK_MODE;
	dir : BOOL;
	tx, last : TIME;
END_VAR

(*
version 1.6	27. jul 2009
programmer 	hugo
tested by		oscat


*)

(* read system timer *)
tx := DWORD_TO_TIME(T_PLC_MS());

(* inputs S1 and S2 are debounced and then decoded for multiple clicks *)
s1e(in := S1, pt := DEBOUNCE_TIME);
s2e(in := S2, pt := DEBOUNCE_TIME);
s1d(in := (s1e.Q AND NOT SINGLE_SWITCH) OR (s1e.Q AND SINGLE_SWITCH AND dir), t_long := CLICK_TIME);
s2d(in := (s2e.Q AND NOT SINGLE_SWITCH) OR (s1e.Q AND SINGLE_SWITCH AND NOT dir), t_long := CLICK_TIME);

(* if d1 and d2 are not toggle clear them to make sure they are only active for oine cycle *)
IF NOT d1_toggle THEN d1 := FALSE; END_IF;
IF NOT d2_toggle THEN d2 := FALSE; END_IF;

(* decode actions *)
IF s1d.tp_LONG THEN
	status := 132;
ELSIF s2d.tp_LONG THEN
	status := 133;
ELSIF  s1d.SINGLE THEN
	IF click_en THEN
		(* if running then we stop otherwise start new direction *)
		IF QU XOR QD THEN
			status := 131;
		ELSE
			status := 134;
			last := tx;
			dir := NOT dir;
		END_IF;
	END_IF;
ELSIF  s2d.SINGLE THEN
	IF click_en THEN
		(* if running then we stop otherwise start new direction *)
		IF QU XOR QD THEN
			status := 131;
		ELSE
			status := 135;
			last := tx;
			dir := NOT dir;
		END_IF;
	END_IF;
ELSIF in THEN
	status := 136;
	last := tx;
ELSIF s1d.DOUBLE THEN
	IF dbl_clk1 THEN
		(* a position need to be set for a double click on S1 *)
		status := 137;
		last := tx;
	ELSE
		(* toggle the output when dbl_clk1 is not active *)
		D1 := NOT D1;
	END_IF;
ELSIF s2d.DOUBLE THEN
	IF dbl_clk2 THEN
		(* a position need to be set for a double click on S2 *)
		status := 138;
		last := tx;
	ELSE
		(* toggle the output when dbl_clk2 is not active *)
		(* in single switch mode we need to toggle d1 instead of d2 *)
		IF single_switch THEN D1 := NOT D1; ELSE D2 := NOT D2; END_IF;
	END_IF;
END_IF;


(* state machine *)
CASE status OF
	0:		(* power up operation *)
			status := 130;

	130:	(* automatic operation standby *)
			IF NOT master_mode THEN
				PO := POS;
				AO := ANG;
			END_IF;
			QU := TRUE;
			QD := TRUE;

	131:	(* manual operation standby *)
			QU := FALSE;
			QD := FALSE;
			PO := POS;
			AO := ANG;
			(* manual mode will be ended when timeout is reached *)
			IF tx - last >= manual_timeout THEN
				status := 130;
			END_IF;

	132:	(* manual operation up *)
			QU := TRUE;
			QD := FALSE;
			PO := POS; AO := ANG;
			last := tx;
			IF NOT s1d.LONG THEN status := 131; dir := NOT dir; END_IF;

	133:	(* manual operation down *)
			QU := FALSE;
			QD := TRUE;
			PO := POS; AO := ANG;
			last := tx;
			IF NOT s2d.LONG THEN	status := 131; dir := NOT dir; END_IF;

	134:	(* manual operation single click up *)
			QU := TRUE;
			QD := FALSE;
			PO := POS; AO := ANG;
			IF tx - last >= max_runtime THEN status := 131; END_IF;

	135:	(* manual operation single click dn *)
			QU := FALSE;
			QD := TRUE;
			PO := POS; AO := ANG;
			IF tx - last >= max_runtime THEN status := 131;	END_IF;

	136:	(* forced input in = true *)
			QU := TRUE;
			QD := TRUE;
			PO := PI; AO := AI;
			IF tx-last >= max_runtime THEN status := 130; END_IF;

	137:	(* double click1 position *)
			QU := TRUE;
			QD := TRUE;
			PO := DBL_POS1;
			AO := DBL_ANG1;
			IF tx - last >= max_runtime THEN status := 131; END_IF;

	138:	(* double click2 position *)
			QU := TRUE;
			QD := TRUE;
			PO := DBL_POS2;
			AO := DBL_ANG2;
			IF tx - last >= max_runtime THEN status := 131; END_IF;

END_CASE;


(* revision history
hm	29. sep 2007	rev 1.0
	original release

hm	6. oct 2007		rev 1.1
	renamed ps and as to po and ao

hm	30. dec 2007	rev 1.2
	added click_timeout variable and function

hm	16. jul. 2008	rev 1.3
	rewirtten code to allow for more functionality
	added single click mode with single_switch.
	added Debounce for inputs S1 and S2
	added double_click functionality

hm	26. sep. 2008	rev 1.4
	corrected an error while POS and ANG was transferred to outputs PO and AO during automatic modes

hm	22. jan 2009	rev 1.5
	added pulse mode for double click outputs
	added automatic mode for IN

hm	27. jul 2009	rev 1.6
	changed status 0 to 130

*)

END_FUNCTION_BLOCK

// POUs/Logic/FF edge triggered/TOGGLE
FUNCTION_BLOCK TOGGLE
VAR_INPUT
	CLK : BOOL;
	rst : BOOL;
END_VAR
VAR_OUTPUT
	Q : BOOL;
END_VAR
VAR
	edge : BOOL;
END_VAR

(*
version 1.1	30. oct. 2008
programmer 	hugo
tested by	oscat

toggle flip flop the output changes state with every rising edge of clk.

*)

IF rst THEN
	q := 0;
ELSIF clk AND NOT edge THEN
	Q := NOT Q;
END_IF;
edge := clk;

(* revision history

hm	13.9.2007		rev 1.0
	original version

hm	30. oct. 2008	rev 1.1
	deleted unnecessary init

*)

END_FUNCTION_BLOCK

// POUs/Building/electrical/CLICK_MODE
FUNCTION_BLOCK CLICK_MODE
VAR_INPUT
	IN : BOOL;
END_VAR
VAR_OUTPUT
	SINGLE : BOOL;
	DOUBLE : BOOL;
	LONG : BOOL;
	TP_LONG : BOOL;
END_VAR
VAR_INPUT CONSTANT
	T_LONG : TIME := t#500ms;
END_VAR
VAR
	Timer : TP;
	cnt : INT;
	last : BOOL;
END_VAR


(*
version 1.0	13. nov. 2008
programmer 	oscat
tested by	hugo

click_mode decodes an input for single, double or long click and sets the corresponding output single, doulbe or long.
the input configures itself to be high or low active depending on which state the input stays longer than t_reconfig.

*)

(* when input goes high start the timer to decode pulses *)
timer(in := IN, PT := T_LONG);
single := FALSE;
double := FALSE;

IF timer.Q THEN
	(* decode pulses while the timer is active *)
	IF NOT in AND last THEN	cnt := cnt + 1; END_IF;
ELSE
	CASE cnt OF
		1 : single := TRUE;
		2 : double := TRUE;
	END_CASE;
	cnt := 0;
END_IF;
last := in;
TP_LONG := NOT timer.Q AND (NOT LONG) AND IN;
LONG := NOT timer.Q AND in;




(* revision history

hm	13. nov. 2008	rev 1.0
	original release

*)

END_FUNCTION_BLOCK

// POUs/Building/Jalousie/BLIND_NIGHT
FUNCTION_BLOCK BLIND_NIGHT
VAR_INPUT
	UP, DN : BOOL;
	S_IN : BYTE;
	PI, AI : BYTE;
	E_NIGHT : BOOL := TRUE;
	E_DAY	: BOOL := TRUE;
	DTIN : DT;
	SUNRISE, SUNSET : TOD;
END_VAR
VAR_INPUT CONSTANT
	sunrise_offset : TIME;
	sunset_offset : TIME;
	night_position : BYTE;
	night_angle : BYTE;
END_VAR
VAR_OUTPUT
	QU, QD : BOOL;
	STATUS : BYTE;
	PO, AO : BYTE;
END_VAR
VAR
	night : BOOL;
	last_night, last_day : DATE;
END_VAR

(*
version 1.2	6 oct 2007
programmer 	hugo
tested by		tobias


*)

IF NOT (up AND dn) AND night THEN
	(* manual operation at night will cancel operation for one night *)
	night := FALSE;
ELSIF (DT_TO_TOD(dtin) > sunset + sunset_offset) AND (last_night < DT_TO_DATE(dtin)) AND NOT night AND e_night THEN
	(* enable night *)
	night := TRUE;
	last_night := DT_TO_DATE(dtin);
ELSIF (DT_TO_TOD(dtin) > sunrise + sunrise_offset) AND (last_day < DT_TO_DATE(dtin)) AND night AND e_day AND (last_night < DT_TO_DATE(dtin)) THEN
	(* disable night *)
	night := FALSE;
	last_day := DT_TO_DATE(dtin);
END_IF;

(* shade at night only in auto mode and enable = true *)
IF UP AND DN AND night THEN
	status := 141;
	po := night_position;
	ao := night_angle;
ELSE
	QU := UP;
	QD := DN;
	po := pi;
	ao := ai;
	status := s_in;
END_IF;


(* revision history
hm	29. sep 2007	rev 1.0
	original version

hm	5. oct 2007		rev 1.1
	added enable input

hm	6. oct 2007		rev 1.2
	added pos and angle inputs and outputs
	night position and angle can now be configured
	any manual operation at night will cancel night operation

*)

END_FUNCTION_BLOCK

// POUs/Building/Jalousie/BLIND_SCENE
FUNCTION_BLOCK BLIND_SCENE
VAR_INPUT
	UP, DN : BOOL;
	S_IN : BYTE;
	PI, AI : BYTE;
	ENABLE : BOOL;
	SWRITE : BOOL;
	SCENE : BYTE;
END_VAR
VAR_OUTPUT
	QU, QD : BOOL;
	STATUS : BYTE;
	PO, AO : BYTE;
END_VAR
VAR RETAIN
	sx : ARRAY[0..15,0..2] OF BYTE;
END_VAR
VAR
	x : BYTE;
END_VAR

(*
version 1.1	29. jan 2008
programmer 	hugo
tested by		tobias


*)

(* delete all bits except the lower 4 of scene *)
x := scene AND 16#0F;

IF enable AND sx[x,2] > 0 AND UP AND DN THEN
	po := sx[x,0];
	ao := sx[x,1];
	status := 160 + x;  (* Status number is 160 to 175 for the 16 scenes *)
	QU := TRUE;
	QD := TRUE;
ELSE
	QU := UP;
	QD := DN;
	status := S_IN;
	po := pi;
	ao := ai;
END_IF;

(* write scene if necessary *)
IF swrite THEN
	status := 176;		(* write scene *)
	sx[x,0] := pi;
	sx[x,1] := ai;
	IF enable THEN sx[x,2] := 1; ELSE sx[x,2] := 0; END_IF; (* if sx[x,2] = 0 the scene is disabled *)
END_IF;


(* revision history
hm	24. oct 2007	rev 1.0
	original release

hm		29.1.2008	rev 1.1
	replaced shr/shl with and for better performance
*)

END_FUNCTION_BLOCK

// POUs/Building/Jalousie/BLIND_SECURITY
FUNCTION_BLOCK BLIND_SECURITY
VAR_INPUT
	UP, DN : BOOL;
	S_IN : BYTE;
	PI, AI : BYTE;
	FIRE : BOOL;
	WIND : BOOL;
	ALARM : BOOL;
	DOOR : BOOL;
	RAIN : BOOL;
END_VAR
VAR_INPUT CONSTANT
	Alarm_UP : BOOL := TRUE;
	WIND_UP :BOOL := TRUE;
	RAIN_UP : BOOL := FALSE;
END_VAR
VAR_OUTPUT
	QU, QD : BOOL;
	STATUS : BYTE;
	PO, AO : BYTE;
END_VAR


(*
version 1.2	12. feb 2008
programmer 	hugo
tested by		tobias


*)

IF Fire THEN
	QU := TRUE;
	QD := FALSE;
	status := 111;
ELSIF Wind THEN
	QU := Wind_up;
	QD := NOT wind_up;
	status := 112;
ELSIF alarm THEN
	QU := Alarm_up;
	QD := NOT Alarm_up;
	status := 113;
ELSIF Door THEN
	QU := TRUE;
	QD := FALSE;
	status := 114;
ELSIF Rain AND NOT (up XOR dn) THEN
	QU := rain_up;
	QD := NOT rain_up;
	status := 115;
ELSE
	QU := UP;
	QD := DN;
	status := S_IN;
	po := pi;
	ao := ai;
END_IF;


(* revision history
hm	29. sep 2007	rev 1.0
	original release

hm	6. oct 2007		rev 1.1
	added pos and angle inputs and outputs
	manual will override rain position
	alarm position can now be configured

hm		12. feb. 2008	rev 1.2
	added config variables rain_up and wind_up
	position for rain and wind is now configurable
*)

END_FUNCTION_BLOCK

// POUs/Building/Jalousie/BLIND_SET
FUNCTION_BLOCK BLIND_SET
VAR_INPUT
	UP, DN : BOOL;
	S_IN : BYTE;
	PI, AI : BYTE;
	IN : BOOL;
	PX, AX : BYTE;
END_VAR
VAR_INPUT CONSTANT
	OVERRIDE_MANUAL : BOOL;
	RESTORE_POSITION : BOOL;
	RESTORE_TIME : TIME := T#60s;
END_VAR
VAR_OUTPUT
	QU, QD : BOOL;
	STATUS : BYTE;
	PO, AO : BYTE;
END_VAR
VAR
	tx: TIME;
	ps: BYTE;
	as: BYTE;
	last: TIME;
END_VAR

(*
version 1.0	27. jul 2009
programmer 	hugo
tested by		oscat

BLIND_SET can be used to force a definite position and angle.
blind_set can be placed close to blind_control for high priority while blind_input must be always at the beginning of the chain with low priority.

*)

(* read system time *)
tx := DWORD_TO_TIME(T_PLC_MS());

(* check inputs *)
IF IN THEN
	IF override_manual OR (UP AND DN) THEN
		status := 178;
	END_IF;
END_IF;

(* state machine *)
CASE STATUS OF
	0: (* power on state *)
		status := S_IN;

	178: (* force values from PX and AX *)
		PO := PX;
		AO := AX;
		QU := TRUE;
		QD := TRUE;
		(* check for end of forced position *)
		IF NOT in THEN
			STATUS := SEL(RESTORE_POSITION, S_IN, 179);
			last := tx;
		END_IF;

	179: (* restore previous position *)
		PO := ps;
		AO := as;
		IF ((PO = PI) AND (AO = AI))  OR tx - last >= RESTORE_TIME THEN
			status := S_IN;
		END_IF;

ELSE
	(* no operation transfer inputs to outputs *)
	PO := PI;
	ps := PI;
	AO := AI;
	as := AI;
	STATUS := S_IN;
	QU := UP;
	QD := DN;
END_CASE;


(* revision history
hm	27. jul 2009	rev 1.0
	original release

*)

END_FUNCTION_BLOCK

// POUs/Building/Jalousie/BLIND_SHADE
FUNCTION_BLOCK BLIND_SHADE
VAR_INPUT
	UP, DN : BOOL;
	S_IN : BYTE;
	PI, AI : BYTE;
	ENABLE : BOOL;
	SUN : BOOL;
END_VAR
VAR_IN_OUT
	CX : calendar;
END_VAR
VAR_INPUT CONSTANT
	sunrise_offset : TIME := T#1h;
	sunset_preset : TIME := T#1h;
	direction : REAL := 180.0;
	angle_offset : REAL := 80.0;
	slat_width : REAL := 80.0;
	Slat_spacing : REAL := 60.0;
	Shade_delay : TIME := T#60s;
	Shade_pos : BYTE;
END_VAR
VAR_OUTPUT
	QU, QD : BOOL;
	STATUS : BYTE;
	PO, AO : BYTE;
END_VAR
VAR
	angle: REAL;
	sun_delay : TOF;
END_VAR

(*
version 1.4	13. mar. 2009
programmer 	hugo
tested by		tobias


*)

(* the input sun is sent through tof which will delay the shade for the time shade_delay *)
sun_delay(IN := sun, PT := shade_delay);

IF UP AND DN AND enable AND sun_delay.Q AND cx.SUN_HOR > direction - angle_offset AND cx.SUN_HOR < direction + angle_offset AND
	DT_TO_TOD(cx.UTC) > cx.SUN_RISE + sunrise_offset AND DT_TO_TOD(cx.UTC) < cx.SUN_SET - sunset_preset THEN
	status := 151;
	QU := UP;
	QD := DN;
	(* position is predefined *)
	po := shade_pos;
	(* shading is active now calculate the slat angle *)
	(* calculate the max angle for the blind *)
	angle := DEG(ATAN(slat_spacing / slat_width));
	(* check if sun angle is between 0 and max angle *)
	IF cx.SUN_VER > 0.0 AND cx.SUN_VER < angle THEN
		angle := cx.SUN_VER + DEG(ACOS(COS(RAD(cx.SUN_VER))*slat_spacing / Slat_width));
		ao := INT_TO_BYTE(LIMIT(0,TRUNC_INT(angle * 2.833333333), 255));
	ELSE
		ao := 255;
	END_IF;
ELSE
	QU := UP;
	QD := DN;
	po := pi;
	ao := ai;
	status := S_IN;
END_IF;

(* revision history
hm	15 oct. 2007	rev 1.0
	original version

hm	19. oct 2007	rev 1.1
	manual mode was not detected because outputs were checked and not inputs UP and DN

hm	24. nov 2007	rev 1.2
	added shade_delay to avoid constant up and down if sun is out parcially

hm	8. feb 2009	rev 1.3
	added shading position shade_pos to be configured
	changed inputs to utilize calendar data structure

hm	13. mar. 2009	rev 1.4
	improved code

*)

END_FUNCTION_BLOCK

// POUs/Building/HLK/BOILER
FUNCTION_BLOCK BOILER
VAR_INPUT
	T_upper : REAL;
	T_lower : REAL;
	Pressure : BOOL := TRUE;
	enable : BOOL := TRUE;
	Req_1 : BOOL;
	Req_2 : BOOL;
	Boost : BOOL;
END_VAR
VAR_INPUT CONSTANT
	t_upper_min : REAL := 50.0;
	t_upper_max : REAL := 60.0;
	T_lower_enable : BOOL;
	T_lower_max : REAL := 60.0;
	T_request_1 : REAL := 70.0;
	T_request_2 : REAL := 50.0;
	T_request_hys : REAL := 5.0;
	T_protect_high : REAL := 80.0;
	T_protect_low : REAL := 10.0;
END_VAR
VAR_OUTPUT
	Heat : BOOL;
	error : BOOL;
	status : BYTE;
END_VAR
VAR
	edge: BOOL;
	boost_mode: BOOL;
	flag_0 : BOOL;
	flag_1: BOOL;
	flag_2: BOOL;
END_VAR

(*
version 1.2	13. mar. 2009
programmer 	hugo
tested by		oscat


this function block controls a hot water boiler. The Boiler can be equipped with two temperature sensors on top and bottom of the tank, T_LOWER_ENABLE must be set to True in this case.
alternatively can BOILER be configured for one (TOP) temperature sensor only (T_LOWER_ENABLE set to False).
A Pressure sensor is used to detect fresh water pressure and disable all heating if there is no water pressure. This input is dset to True by default, so if it is not used it can simply be left open.
A enable input enables the hot water heating while it is set to True. alternatively can a Ture on Req_1 or Req_2 start the heating to predefined temperatures during setup.
A low to high edge on the boost input will start heating imediately until T_upper_max is reached, it can be used to generate extra hot water when needed.

*)

(* read sensors and check for valid data *)
IF t_upper > t_protect_high THEN
	status := 1;
	heat := FALSE;
	error := TRUE;
ELSIF t_upper < t_protect_low THEN
	status := 2;
	heat :=	TRUE;
	error := TRUE;
ELSIF t_lower > T_protect_high AND t_lower_enable THEN
	status := 3;
	heat := FALSE;
	error := TRUE;
ELSIF t_lower < t_protect_low AND t_lower_enable THEN
	status := 4;
	heat := TRUE;
	error := TRUE;
ELSIF NOT pressure THEN
	status := 5;
	heat := FALSE;
	error := TRUE;
ELSIF req_1 OR req_2 OR enable OR boost THEN
	error := FALSE;

	(* determine if heat needs to be turned on *)
	IF boost AND NOT edge AND t_upper < t_upper_max THEN
		status := 101;
		heat := TRUE;
		boost_mode := TRUE;
	ELSIF enable AND t_upper < T_upper_min THEN
		status := 102;
		heat := TRUE;
	ELSIF req_1 AND t_upper < T_request_1 THEN
		status := 103;
		heat := TRUE;
	ELSIF req_2 AND t_upper < t_request_2 THEN
		status := 104;
		heat := TRUE;
	END_IF;

	(* determine the shut off temperature *)
	IF heat THEN
		IF (enable OR boost_mode) THEN
			flag_0 := TRUE;
			IF T_lower_enable AND T_lower > T_lower_max THEN
				flag_0 := boost_mode := FALSE;
			ELSIF NOT T_lower_enable AND T_upper > T_upper_max THEN
				flag_0 := boost_mode := FALSE;
			END_IF;
		ELSE
			flag_0 := FALSE;
		END_IF;
		flag_1 := (req_1 AND T_upper > T_request_1 + T_request_hys) AND req_1;
		flag_2 := (req_2 AND T_upper > T_request_2 + T_request_hys) AND req_2;

		(* shut off heat if no longer needed *)
		heat := flag_0 OR flag_1 OR flag_2;
		IF heat = FALSE THEN status := 100; END_IF;
	END_IF;
ELSE
	status := 100;
	heat := FALSE;
	error := FALSE;
END_IF;
edge := boost;


(* revision history
hm	27. feb. 2007	rev 1.0
	original version

hm	16. oct. 2008	rev 1.1
	improved performance

hm	13. mar. 2009	rev 1.2
	real constants updated to new systax using dot
	replaced double assignments
*)

END_FUNCTION_BLOCK

// POUs/Buffer Management/BUFFER_COMP
FUNCTION BUFFER_COMP : INT
VAR_INPUT
	PT1 : POINTER TO ARRAY[0..32767] OF BYTE;
	SIZE1 : INT;
	PT2 : POINTER TO ARRAY[0..32767] OF BYTE;
	SIZE2 : INT;
	START : INT;
END_VAR
VAR
	i, j, end : INT;
END_VAR

(*
version 1.0	14. nov. 2008
programmer 	hugo
tested by	oscat


 
*)

(* search for first character match *)
IF size2 <= size1 THEN
	end := size1 - size2;
	FOR i := START TO end DO
		IF PT1^[i] = PT2^[0] THEN
			(* first character matches, now compare rest of array *)
			j := 1;
			WHILE j < size2 DO
				IF pt2^[j] <> pt1^[j+i] THEN EXIT; END_IF;
				j := j + 1;
			END_WHILE;
			(* when J > size2 a match was found return the position i in buffer1 *)
			IF j = size2 THEN
				BUFFER_COMP := i;
				RETURN;
			END_IF;
		END_IF;
	END_FOR;
END_IF;
BUFFER_COMP := -1;


(*
hm 	14. nov. 2008	rev 1.0
	original version

*)

END_FUNCTION

// POUs/Buffer Management/BUFFER_SEARCH
FUNCTION BUFFER_SEARCH : INT
VAR_INPUT
	PT : POINTER TO ARRAY[0..32767] OF BYTE;
	SIZE : UINT;
	STR : STRING(STRING_LENGTH);
	POS : INT;
	IGN : BYTE;
END_VAR
VAR
	ps : POINTER TO ARRAY[0..255] OF BYTE;
	i: INT;
	end: INT;
	k: INT;
	lx: INT;
END_VAR


(*
version 1.2	13. may. 2008
programmer 	hugo
tested by	oscat

this function will search for a string STR in an array of byte starting at position pos.
the function needs to be called:	buffer_search(adr("array"),sizeof("array"), STR, POS, IGN);
because this function works with pointers its very time efficient and it needs no extra memory.
The function returns the position of the first character of the string in the array if found.
a 0 is returned if the string is not found in the array.
The parameter IGN specifies a wildcard character in the search string.

*)

ps := ADR(str);
lx := LEN(str);
end := UINT_TO_INT(size) - lx;
lx := lx - 1;
FOR i := pos TO end DO
	FOR k := 0 TO lx DO
		IF (ps^[k] <> ign) AND (ps^[k] <> pt^[i+k]) THEN EXIT; END_IF;
	END_FOR;
	IF k > lx THEN
		BUFFER_SEARCH := i;
		RETURN;
	END_IF;
END_FOR;
BUFFER_SEARCH := 0;


(* revision History

hm 5. mar. 2008	rev 1.0
	original version

hm	16. mar. 2008	rev 1.1
	chaged type of input size to uint

hm	13. may. 2008	rev 1.2
	changed type of pointer to array[1..32767]
	changed size of string to STRING_LENGTH

*)

END_FUNCTION

// POUs/Buffer Management/BUFFER_TO_STRING
FUNCTION BUFFER_TO_STRING : STRING(STRING_LENGTH)
VAR_INPUT
	PT : POINTER TO ARRAY[0..32767] OF BYTE;
	SIZE : UINT;
	START : UINT;
	STOP : UINT;
END_VAR
VAR
	ps : POINTER TO BYTE;
	i : UINT;
	stp: UINT;
	sta: UINT;
END_VAR


(*
version 1.4	23. mar. 2009
programmer 	hugo
tested by	oscat

this function will retrieve a string from an array of byte starting at position start and stop at position stop.
the function needs to be called:	buffer_TO_String(adr("array"),sizeof("array"), start, stop);
because this function works with pointers its very time efficient and it needs no extra memory.

*)

ps := ADR(BUFFER_TO_STRING);
sta :=MIN(start, size);
stp := MIN(stop, size);
(* check for maximum string_length *)
IF UINT_TO_INT(stp - sta + 1) >= STRING_LENGTH THEN
	stp := sta + INT_TO_UINT(STRING_LENGTH) - 1;
END_IF;

FOR i := sta TO stp DO
	ps^ := pt^[i];
	ps := ps + 1;
END_FOR;

(* terminate the string *)
ps^ := 0;



(* revision History
hm 	5. mar. 2008	rev 1.0
	original version

hm	16. mar. 2008	rev 1.1
	changed type of input size to uint

hm	13. may. 2008	rev 1.2
	changed type of pointer to array[0..32767]
	changed size of string to STRING_LENGTH

hm	12. jun. 2008	rev 1.3
	check for pointer overrun
	change input start and stop to uint
	added type conversions to avoid warnings under codesys 3.0

hm	23. mar. 2009	rev 1.4
	avoid writing to input stop
*)

END_FUNCTION

// POUs/Logic/gate logic/BYTE_OF_BIT
FUNCTION BYTE_OF_BIT : BYTE
VAR_INPUT
	B0:BOOL;
	B1:BOOL;
	B2:BOOL;
	B3:BOOL;
	B4:BOOL;
	B5:BOOL;
	B6:BOOL;
	B7:BOOL;
END_VAR


(*
version 1.1	 18. feb 2006
programmer 	hugo
tested by		tobias

this function creates a byte from 8 individual bits

*)

Byte_of_bit := SHL(SHL(SHL(SHL(SHL(SHL(SHL(BOOL_TO_BYTE(B7),1) OR BOOL_TO_BYTE(B6),1) OR BOOL_TO_BYTE(B5),1) OR BOOL_TO_BYTE(B4),1)
	OR BOOL_TO_BYTE(B3),1) OR BOOL_TO_BYTE(B2),1) OR BOOL_TO_BYTE(B1),1) OR BOOL_TO_BYTE(B0);


(* revision history

hm	4. aug 2006		rev 1.0
	original version

hm	18. feb. 2008	rev 1.1
	improved performance

*)

END_FUNCTION

// POUs/Logic/gate logic/BYTE_OF_DWORD
FUNCTION BYTE_OF_DWORD : BYTE
VAR_INPUT
	in : DWORD;
	N : BYTE;
END_VAR


(*
version 1.2	30. oct. 2008
programmer 	hugo
tested by	oscat

this function extracts a single byte from the nth position from right (right is lowest byte) 
the lower byte (starting with Bit0 from in) is selected with N=0.
*)

BYTE_OF_DWORD := DWORD_TO_BYTE(SHR(in,SHL(n,3)));

(* revision history
hm	17. jan 2007	rev 1.0
	original version

hm	2. jan 2008		rev 1.1
	improved performance

hm	30. oct. 2008	rev 1.2
	improved performance
*)

END_FUNCTION

// POUs/Logic/gate logic/BYTE_TO_BITS
FUNCTION_BLOCK BYTE_TO_BITS
VAR_INPUT
	IN: BYTE;
END_VAR
VAR_OUTPUT
	B0: BOOL;
	B1: BOOL;
	B2: BOOL;
	B3: BOOL;
	B4: BOOL;
	B5: BOOL;
	B6: BOOL;
	B7: BOOL;
END_VAR


(*
version 1.1	16. mar. 2008
programmer 	hugo
tested by		tobias

this Function Block extracts the 8 Bits from a byte


*)

B0 := IN.0;
B1 := IN.1;
B2 := IN.2;
B3 := IN.3;
B4 := IN.4;
B5 := IN.5;
B6 := IN.6;
B7 := IN.7;

(* revision history
hm		4. aug 2006	rev 1.0
	original version

hm		16. mar 2008	rev 1.1
	renamed from byte_to_bit to byte_to_bits for compatibility reasons

*)

END_FUNCTION_BLOCK

// POUs/Engineering/signal processing/BYTE_TO_RANGE
FUNCTION BYTE_TO_RANGE : REAL
VAR_INPUT
	X : BYTE;
	low : REAL;
	high : REAL;
END_VAR


(*
version 1.0	9. jan 2008
programmer 	hugo
tested by		tobias

Byte_to_Range converts a Byte into a real between low and high.

*)

BYTE_TO_RANGE := (high - low) * X / 255.0 + low;


(* revision history
hm	9. jan 2008		rev 1.0
	original version

*)

END_FUNCTION

// POUs/String/BYTE_TO_STRB
FUNCTION BYTE_TO_STRB : STRING(8)
VAR_INPUT
	IN : BYTE;
END_VAR
VAR
	i: INT;
	pt : POINTER TO BYTE;
END_VAR

(*
version 1.3	20. jun. 2008
programmer 	hugo
tested by	oscat

BYTE_TO_STRINGB converts a Byte to a String of Bits represented by '0' and '1' s.
The lowest order bit will be on the right and the high order bit on the left.

*)

(* pointer für die ausgabe ermitteln *)
pt := ADR(BYTE_TO_STRB);
(* die 8 ausgabecharacter ermitteln und schreiben *)
FOR i := 1 TO 8 DO
	pt^ := BOOL_TO_BYTE(in.7) + 48;
	in := SHL(in,1);
	pt := pt + 1;
END_FOR;

(* der ausgabestring muss noch mit 0 abgeschlossen werden *)
pt^ := 0;

(* code before rev 1.1
FOR i := 1 TO 8 DO
	IF in.0 = 0 THEN temp := CONCAT('0', temp); ELSE temp := CONCAT('1', temp); END_IF;
	in := SHR(in, 1);
END_FOR;
BYTE_TO_STRB := temp;
*)


(* revision history

hm		9.6.2007	rev 1.0		
	original version 

hm	15. dec 2007	rev 1.1
	inprooved code for higher performance

hm	29. mar. 2008	rev 1.2
	changed STRING to STRING(8)

hm	20. jun. 2008	rev 1.3
	performance improvement

*)

END_FUNCTION

// POUs/String/BYTE_TO_STRH
FUNCTION BYTE_TO_STRH : STRING(2)
VAR_INPUT
	IN : BYTE;
END_VAR
VAR
	temp : BYTE;
	PT : POINTER TO BYTE;
END_VAR

(*
version 1.3	29 mar. 2008
programmer 	hugo
tested by		tobias

BYTE_TO_STRINGH converts a Byte to a String of Hexadecimal represented by '0' .. '9' and 'A' .. 'F'.
The lowest order Character will be on the right and the high order Character on the left.

*)

(* read pointer to output string *)
PT := ADR(BYTE_TO_STRH);
(* calculate high order hex value *)
temp := SHR(in,4);
(* convert value to hex character *)
IF temp <= 9 THEN temp := temp + 48; ELSE temp := temp + 55; END_IF;
(* write friat character to output string *)
PT^ := temp;
(* calculate low order hex value *)
temp := in AND 2#00001111;
IF temp <= 9 THEN temp := temp + 48; ELSE temp := temp + 55; END_IF;
(* increment pointer and wirte low order character *)
pt := pt + 1;
pt^ := temp;
(* set pointer at the end of the output string and close the string with 0 *)
pt := pt + 1;
pt^:= 0;


(* code before rev 1.2
FOR i := 1 TO 2 DO
	X := in AND 2#1111;
	IF X <= 9 THEN X := X + 48; ELSE X := X + 55; END_IF;
	Cx := CHR(X);
	temp := CONCAT(Cx, temp);
	in := SHR(in,4);
END_FOR;
BYTE_TO_STRH := temp;
*)

(* revision history

hm	9.6.2007		rev 1.0		
	original version 

hm	11.9.2007		rev 1.1		
	changed coding for compatibility with twincat, under twincat concat cannot have a function as argument.	

hm	15 dec 2007		REV 1.2
	changed code for higher performance

hm	29. mar. 2008	rev 1.3
	changed STRING to STRING(2)
*)

END_FUNCTION

// POUs/Engineering/conversion/C_TO_F
FUNCTION C_TO_F : REAL
VAR_INPUT
	celsius : REAL;
END_VAR


(*
version 1.1	11. mar. 2009
programmer 	hugo
tested by		tobias

this function converts celsius  to fahrenheit 

*)

C_TO_F := celsius * 1.8 + 32.0;


(* revision history

hm	4. aug. 2006	rev 1.0
	original version

hm	11. mar. 2009	rev 1.1
	real constants updated to new systax using dot

*)

END_FUNCTION

// POUs/Engineering/conversion/C_TO_K
FUNCTION C_TO_K : REAL
VAR_INPUT
	Celsius : REAL;
END_VAR


(*
version 1.0	4 dec 2006
programmer 	hugo
tested by		tobias

this function converts celsius to kelvin
*)

C_TO_K := Celsius - 273.15;

(* revision history

hm	4. aug 2006	rev 1.0
	original version

*)

END_FUNCTION

// POUs/Mathematical/Complex/CABS
FUNCTION CABS : REAL
VAR_INPUT
	X : complex;
END_VAR


(*
version 1.0	21 feb 2008
programmer 	hugo
tested by	oscat

this function the aboslute value of a complex number

*)

CABS := HYPOT(x.re, x.im);


(* revision history
hm	21. feb 2008	rev 1.0
	original version

*)

END_FUNCTION

// POUs/Mathematical/HYPOT
FUNCTION HYPOT : REAL
VAR_INPUT
	X : REAL;
	Y : REAL;
END_VAR


(*
version 1.0	21 feb 2008
programmer 	hugo
tested by	oscat

this function calculates the pythagorean function

*)

HYPOT := SQRT(x*x + y*y);


(* revision history
hm	21. feb 2008	rev 1.0
	original version

*)

END_FUNCTION

// POUs/Mathematical/Complex/CACOS
FUNCTION CACOS : complex
VAR_INPUT
	X : complex;
END_VAR
VAR
	Y : complex;
END_VAR

(*
version 1.0	21 feb 2008
programmer 	hugo
tested by	oscat

this function calculates the arcus cosinus function of a complex number

*)

y := CACOSH(x);
CACOS.re := y.im;
CACOS.im := -y.re;



(* revision history
hm	21. feb 2008	rev 1.0
	original version


*)

END_FUNCTION

// POUs/Mathematical/Complex/CACOSH
FUNCTION CACOSH : complex
VAR_INPUT
	X : complex;
END_VAR
VAR
	Y : complex;
END_VAR

(*
version 1.0	21 feb 2008
programmer 	hugo
tested by	oscat

this function calculates the hyperbolic arcus cosinus function of a complex number

*)

y.re := (X.re - X.im)*(X.re + X.im) - 1.0;
y.im := 2.0 * X.re * X.im;
y    := CSQRT(y);
y.re := y.re + x.re;
y.im := y.im + x.im;
CACOSH  := CLOG(y);



(* revision history
hm	21. feb 2008	rev 1.0
	original version


*)

END_FUNCTION

// POUs/Mathematical/Complex/CSQRT
FUNCTION CSQRT : complex
VAR_INPUT
	X : complex;
END_VAR
VAR
	temp : REAL;
END_VAR

(*
version 1.0	21 feb 2008
programmer 	hugo
tested by	oscat

this function calculates the complex sqare root

*)

temp := HYPOT(x.re, x.im);
CSQRT.re :=  SQRT(0.5 * (temp + x.re));
CSQRT.im :=  sgn(x.im) * SQRT(0.5 * (temp - x.re));


(* revision history
hm	21. feb 2008	rev 1.0
	original version

*)

END_FUNCTION

// POUs/Mathematical/SGN
FUNCTION SGN : INT
VAR_INPUT
	X : REAL;
END_VAR


(*
version 1.1	11. nov. 2008
programmer 	hugo
tested by	tobias

sgn returns 0 when X = 0 , -1 when X < 1 and +1 when X > 1

*)

IF X > 0 THEN
	SGN := 1;
ELSIF X < 0 THEN
	SGN := -1;
ELSE
	SGN := 0;
END_IF;



(* revision histroy
hm	16. oct 2007	rev 1.0
	original version

hm	11. nov 2007	rev 1.1
	changed type of function from real to int

*)

END_FUNCTION

// POUs/Mathematical/Complex/CLOG
FUNCTION CLOG : complex
VAR_INPUT
	X : complex;
END_VAR


(*
version 1.1	20. apr. 2008
programmer 	hugo
tested by	oscat

this function calculates the complex natural (base e) logarithm

*)

CLOG.re := LN(HYPOT(X.re, X.im));
CLOG.im := ATAN2(X.im, X.re);


(* revision history
hm	21. feb 2008	rev 1.0
	original version

hm	20. apr. 2008	rev 1.1
	use ATAN2 instead of ATAN
*)

END_FUNCTION

// POUs/Mathematical/Complex/CADD
FUNCTION CADD : complex
VAR_INPUT
	X, Y : complex;
END_VAR


